RoboDK station: colorBars_ROR.rdk

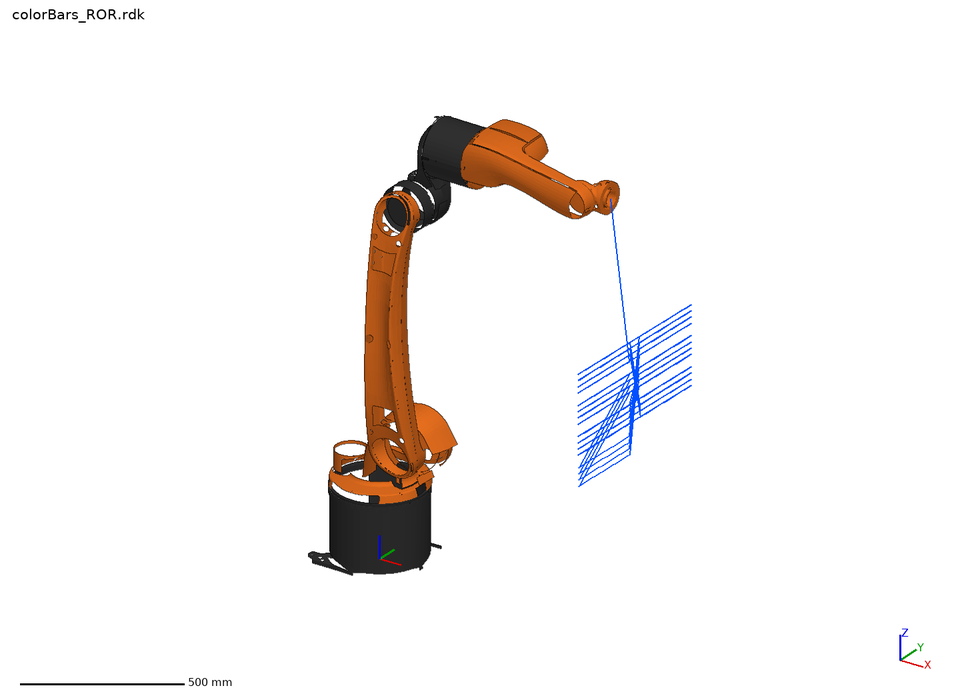
[picture v0: the station drawn from its stored meshes, robots at their saved joint values, targets as dots, program paths as lines]
Station pv_f053_run_on_robot (saved by RoboDK 5.4.1). Poses are relative to the parent item; angles as X-Y-Z fixed-axis rotations.
  - frame KR 8 1620 ARC HW Base at (0, 0, 0) mm
    - robot KR 8 1620 ARC HW: 6 axes
        modified DH rows (alpha deg, a mm, theta deg, d mm): 0, 0, 0, 450; -90, 150, 0, 0; 0, 810, -90, 0; -90, 200, 0, 630; 90, 0, 0, 0; -90, 0, 180, 80
        joint limits [-170, -185, -120, -165, -115, -350] to [170, 65, 180, 165, 140, 350]; home [0, -90, 90, 0, 0, 0]; saved at [0, -90, 90, 0, 0, 0]
      - tool fbx_0_slot_00_fo1_roundShape_outPaintBrush, TCP at (-4.14, -15.45, 32) mm
      - tool fbx_1_slot_01_fo2_roundShape_outPaintBrush, TCP at (-15.45, -4.14, 32) mm
      - tool fbx_2_slot_02_fo3_roundShape_outPaintBrush, TCP at (-11.31, 11.31, 32) mm
      - tool fbx_3_slot_03_fo4_roundShape_outPaintBrush, TCP at (4.14, 15.45, 32) mm
      - tool fbx_4_slot_04_fo5_roundShape_outPaintBrush, TCP at (15.45, 4.14, 32) mm
      - tool fbx_5_slot_05_fo6_roundShape_outPaintBrush, TCP at (11.31, -11.31, 32) mm
  - frame ax_frame at (0, 0, 0) mm
    - target home_approach (joint target) at (860, 0, 1460) mm, rotated rx 0 ry 90 rz 0 deg; joints [0, -89.818, 101.483, 0, -11.665, 0] of KR 8 1620 ARC HW
  - program pv_f053_00 (1123 instructions, listed below)
  - frame pv_f053_00_frame at (0, 0, 0) mm
    - target init_t0 (Cartesian target) at (979.8, -18.27, 823.95) mm, rotated rx 136.82 ry 86.87 rz 134.63 deg; joints [1.647, -75.367, 132.098, -0.612, -54.447, -1.81] of KR 8 1620 ARC HW
    - target stk_p0_s0_t0 (Cartesian target) at (979.8, -18.27, 823.95) mm, rotated rx 136.82 ry 86.87 rz 134.63 deg; joints [1.647, -75.367, 132.098, -0.612, -54.447, -1.81] of KR 8 1620 ARC HW
    - target stk_p0_s0_t0 (Cartesian target) at (979.8, -18.27, 823.95) mm, rotated rx 136.82 ry 86.87 rz 134.63 deg; joints [1.647, -75.367, 132.098, -0.612, -54.447, -1.81] of KR 8 1620 ARC HW
    - target stk_p0_s0_t1 (Cartesian target) at (980.02, -7.71, 824.07) mm, rotated rx 132.07 ry 86.58 rz 129.48 deg; joints [0.893, -75.374, 132.102, -2.02, -54.454, -1.429] of KR 8 1620 ARC HW
    - target stk_p0_s0_t2 (Cartesian target) at (980.24, 2.85, 824.19) mm, rotated rx 128.07 ry 86.28 rz 125.08 deg; joints [0.139, -75.372, 132.093, -3.428, -54.473, -1.049] of KR 8 1620 ARC HW
    - target stk_p0_s0_t3 (Cartesian target) at (980.46, 13.4, 824.32) mm, rotated rx 124.68 ry 85.96 rz 121.29 deg; joints [-0.614, -75.361, 132.07, -4.835, -54.503, -0.67] of KR 8 1620 ARC HW
    - target stk_p0_s0_t4 (Cartesian target) at (980.68, 23.96, 824.44) mm, rotated rx 121.8 ry 85.63 rz 118.01 deg; joints [-1.367, -75.34, 132.034, -6.239, -54.545, -0.292] of KR 8 1620 ARC HW
    - target stk_p0_s0_t5 (Cartesian target) at (980.89, 34.52, 824.56) mm, rotated rx 119.33 ry 85.29 rz 115.14 deg; joints [-2.12, -75.31, 131.985, -7.642, -54.598, 0.085] of KR 8 1620 ARC HW
    - target stk_p0_s0_t6 (Cartesian target) at (981.11, 45.08, 824.69) mm, rotated rx 117.2 ry 84.94 rz 112.61 deg; joints [-2.871, -75.27, 131.923, -9.04, -54.663, 0.46] of KR 8 1620 ARC HW
    - target stk_p0_s0_t7 (Cartesian target) at (981.33, 55.64, 824.81) mm, rotated rx 115.34 ry 84.59 rz 110.35 deg; joints [-3.621, -75.221, 131.848, -10.435, -54.74, 0.832] of KR 8 1620 ARC HW
    - target stk_p0_s0_t8 (Cartesian target) at (981.55, 66.2, 824.94) mm, rotated rx 113.72 ry 84.23 rz 108.33 deg; joints [-4.369, -75.163, 131.759, -11.825, -54.828, 1.201] of KR 8 1620 ARC HW
    - target stk_p0_s0_t9 (Cartesian target) at (981.77, 76.75, 825.06) mm, rotated rx 112.28 ry 83.87 rz 106.49 deg; joints [-5.115, -75.095, 131.658, -13.21, -54.927, 1.567] of KR 8 1620 ARC HW
    - target stk_p0_s0_t10 (Cartesian target) at (981.99, 87.31, 825.18) mm, rotated rx 111.01 ry 83.51 rz 104.82 deg; joints [-5.859, -75.019, 131.543, -14.588, -55.037, 1.929] of KR 8 1620 ARC HW
    - target stk_p0_s0_t11 (Cartesian target) at (982.21, 97.87, 825.31) mm, rotated rx 109.87 ry 83.14 rz 103.28 deg; joints [-6.601, -74.933, 131.415, -15.961, -55.158, 2.288] of KR 8 1620 ARC HW
    - target stk_p0_s0_t12 (Cartesian target) at (982.43, 108.43, 825.43) mm, rotated rx 108.85 ry 82.77 rz 101.87 deg; joints [-7.339, -74.838, 131.274, -17.325, -55.289, 2.642] of KR 8 1620 ARC HW
    - target stk_p0_s0_t13 (Cartesian target) at (982.65, 118.99, 825.55) mm, rotated rx 107.93 ry 82.4 rz 100.55 deg; joints [-8.075, -74.733, 131.12, -18.682, -55.431, 2.991] of KR 8 1620 ARC HW
    - target stk_p0_s0_t14 (Cartesian target) at (982.87, 129.55, 825.68) mm, rotated rx 107.09 ry 82.03 rz 99.32 deg; joints [-8.808, -74.62, 130.953, -20.031, -55.583, 3.336] of KR 8 1620 ARC HW
    - target stk_p0_s0_t15 (Cartesian target) at (983.09, 140.11, 825.8) mm, rotated rx 106.33 ry 81.66 rz 98.16 deg; joints [-9.537, -74.498, 130.773, -21.371, -55.745, 3.675] of KR 8 1620 ARC HW
    - target stk_p0_s0_t16 (Cartesian target) at (983.31, 150.66, 825.92) mm, rotated rx 105.64 ry 81.29 rz 97.07 deg; joints [-10.262, -74.367, 130.58, -22.701, -55.917, 4.009] of KR 8 1620 ARC HW
    - target stk_p0_s0_t17 (Cartesian target) at (983.53, 161.22, 826.05) mm, rotated rx 105 ry 80.91 rz 96.04 deg; joints [-10.984, -74.228, 130.374, -24.022, -56.098, 4.338] of KR 8 1620 ARC HW
    - target stk_p0_s0_t18 (Cartesian target) at (983.75, 171.78, 826.17) mm, rotated rx 104.42 ry 80.54 rz 95.06 deg; joints [-11.701, -74.08, 130.155, -25.332, -56.289, 4.66] of KR 8 1620 ARC HW
    - target stk_p0_s0_t19 (Cartesian target) at (983.96, 182.34, 826.29) mm, rotated rx 103.88 ry 80.17 rz 94.13 deg; joints [-12.414, -73.923, 129.923, -26.632, -56.488, 4.977] of KR 8 1620 ARC HW
    - target stk_p0_s0_t20 (Cartesian target) at (984.18, 192.9, 826.42) mm, rotated rx 103.38 ry 79.79 rz 93.24 deg; joints [-13.123, -73.758, 129.679, -27.92, -56.696, 5.288] of KR 8 1620 ARC HW
    - target stk_p0_s0_t21 (Cartesian target) at (984.4, 203.46, 826.54) mm, rotated rx 102.91 ry 79.42 rz 92.38 deg; joints [-13.826, -73.584, 129.422, -29.198, -56.912, 5.593] of KR 8 1620 ARC HW
    - target stk_p0_s0_t22 (Cartesian target) at (984.62, 214.01, 826.67) mm, rotated rx 102.48 ry 79.05 rz 91.56 deg; joints [-14.525, -73.402, 129.152, -30.463, -57.136, 5.891] of KR 8 1620 ARC HW
    - target stk_p0_s0_t23 (Cartesian target) at (984.84, 224.57, 826.79) mm, rotated rx 102.08 ry 78.67 rz 90.76 deg; joints [-15.219, -73.212, 128.87, -31.717, -57.368, 6.183] of KR 8 1620 ARC HW
    - target stk_p0_s0_t24 (Cartesian target) at (985.06, 235.13, 826.91) mm, rotated rx 101.7 ry 78.3 rz 90 deg; joints [-15.907, -73.014, 128.575, -32.958, -57.608, 6.469] of KR 8 1620 ARC HW
    - target stk_p0_s0_t25 (Cartesian target) at (985.28, 245.69, 827.04) mm, rotated rx 101.35 ry 77.93 rz 89.26 deg; joints [-16.59, -72.808, 128.268, -34.186, -57.855, 6.749] of KR 8 1620 ARC HW
    - target stk_p0_s1_t0 (Cartesian target) at (973.22, -335.02, 820.24) mm, rotated rx -102.56 ry 80.25 rz -92.87 deg; joints [22.967, -71.014, 125.959, 38.741, -59.048, -11.564] of KR 8 1620 ARC HW
    - target stk_p0_s1_t0 (Cartesian target) at (973.22, -335.02, 820.24) mm, rotated rx -102.56 ry 80.25 rz -92.87 deg; joints [22.967, -71.014, 125.959, 38.741, -59.048, -11.564] of KR 8 1620 ARC HW
    - target stk_p0_s1_t1 (Cartesian target) at (973.44, -324.47, 820.36) mm, rotated rx -103.11 ry 80.62 rz -93.8 deg; joints [22.327, -71.275, 126.345, 37.585, -58.778, -11.319] of KR 8 1620 ARC HW
    - target stk_p0_s1_t2 (Cartesian target) at (973.66, -313.91, 820.49) mm, rotated rx -103.7 ry 80.99 rz -94.78 deg; joints [21.681, -71.529, 126.719, 36.415, -58.514, -11.068] of KR 8 1620 ARC HW
    - target stk_p0_s1_t3 (Cartesian target) at (973.88, -303.35, 820.61) mm, rotated rx -104.33 ry 81.36 rz -95.8 deg; joints [21.028, -71.776, 127.08, 35.233, -58.255, -10.811] of KR 8 1620 ARC HW
    - target stk_p0_s1_t4 (Cartesian target) at (974.1, -292.79, 820.73) mm, rotated rx -105.03 ry 81.73 rz -96.89 deg; joints [20.37, -72.016, 127.43, 34.037, -58.003, -10.548] of KR 8 1620 ARC HW
    - target stk_p0_s1_t5 (Cartesian target) at (974.32, -282.23, 820.86) mm, rotated rx -105.8 ry 82.1 rz -98.05 deg; joints [19.705, -72.248, 127.767, 32.829, -57.757, -10.279] of KR 8 1620 ARC HW
    - target stk_p0_s1_t6 (Cartesian target) at (974.53, -271.67, 820.98) mm, rotated rx -106.64 ry 82.46 rz -99.28 deg; joints [19.035, -72.474, 128.093, 31.608, -57.517, -10.004] of KR 8 1620 ARC HW
    - target stk_p0_s1_t7 (Cartesian target) at (974.75, -261.11, 821.11) mm, rotated rx -107.56 ry 82.83 rz -100.59 deg; joints [18.359, -72.691, 128.406, 30.375, -57.285, -9.722] of KR 8 1620 ARC HW
    - target stk_p0_s1_t8 (Cartesian target) at (974.97, -250.56, 821.23) mm, rotated rx -108.59 ry 83.19 rz -102.01 deg; joints [17.677, -72.901, 128.706, 29.129, -57.059, -9.435] of KR 8 1620 ARC HW
    - target stk_p0_s1_t9 (Cartesian target) at (975.19, -240, 821.35) mm, rotated rx -109.73 ry 83.56 rz -103.55 deg; joints [16.99, -73.103, 128.995, 27.872, -56.841, -9.142] of KR 8 1620 ARC HW
    - target stk_p0_s1_t10 (Cartesian target) at (975.41, -229.44, 821.48) mm, rotated rx -111.02 ry 83.92 rz -105.23 deg; joints [16.297, -73.297, 129.271, 26.602, -56.631, -8.842] of KR 8 1620 ARC HW
    - target stk_p0_s1_t11 (Cartesian target) at (975.63, -218.88, 821.6) mm, rotated rx -112.46 ry 84.28 rz -107.07 deg; joints [15.6, -73.483, 129.534, 25.321, -56.429, -8.536] of KR 8 1620 ARC HW
    - target stk_p0_s1_t12 (Cartesian target) at (975.85, -208.32, 821.72) mm, rotated rx -114.1 ry 84.63 rz -109.1 deg; joints [14.897, -73.661, 129.785, 24.029, -56.235, -8.224] of KR 8 1620 ARC HW
    - target stk_p0_s1_t13 (Cartesian target) at (976.07, -197.76, 821.85) mm, rotated rx -115.97 ry 84.98 rz -111.37 deg; joints [14.19, -73.83, 130.023, 22.726, -56.05, -7.907] of KR 8 1620 ARC HW
    - target stk_p0_s1_t14 (Cartesian target) at (976.29, -187.21, 821.97) mm, rotated rx -118.12 ry 85.32 rz -113.92 deg; joints [13.478, -73.992, 130.249, 21.413, -55.874, -7.583] of KR 8 1620 ARC HW
    - target stk_p0_s1_t15 (Cartesian target) at (976.51, -176.65, 822.09) mm, rotated rx -120.61 ry 85.66 rz -116.81 deg; joints [12.762, -74.144, 130.461, 20.089, -55.707, -7.254] of KR 8 1620 ARC HW
    - target stk_p0_s1_t16 (Cartesian target) at (976.73, -166.09, 822.22) mm, rotated rx -123.52 ry 85.99 rz -120.11 deg; joints [12.041, -74.289, 130.662, 18.756, -55.549, -6.919] of KR 8 1620 ARC HW
    - target stk_p0_s1_t17 (Cartesian target) at (976.95, -155.53, 822.34) mm, rotated rx -126.94 ry 86.3 rz -123.92 deg; joints [11.317, -74.424, 130.849, 17.414, -55.4, -6.579] of KR 8 1620 ARC HW
    - target stk_p0_s1_t18 (Cartesian target) at (977.17, -144.97, 822.46) mm, rotated rx -130.98 ry 86.61 rz -128.36 deg; joints [10.589, -74.551, 131.023, 16.063, -55.262, -6.234] of KR 8 1620 ARC HW
    - target stk_p0_s1_t19 (Cartesian target) at (977.39, -134.41, 822.59) mm, rotated rx -135.78 ry 86.89 rz -133.56 deg; joints [9.857, -74.67, 131.185, 14.704, -55.134, -5.883] of KR 8 1620 ARC HW
    - target stk_p0_s1_t20 (Cartesian target) at (977.6, -123.86, 822.71) mm, rotated rx -141.48 ry 87.14 rz -139.67 deg; joints [9.122, -74.779, 131.333, 13.337, -55.016, -5.529] of KR 8 1620 ARC HW
    - target stk_p0_s1_t21 (Cartesian target) at (977.82, -113.3, 822.84) mm, rotated rx -148.23 ry 87.36 rz -146.81 deg; joints [8.384, -74.879, 131.469, 11.964, -54.909, -5.17] of KR 8 1620 ARC HW
    - target stk_p0_s1_t22 (Cartesian target) at (978.04, -102.74, 822.96) mm, rotated rx -156.09 ry 87.54 rz -155.07 deg; joints [7.643, -74.97, 131.591, 10.583, -54.812, -4.807] of KR 8 1620 ARC HW
    - target stk_p0_s1_t23 (Cartesian target) at (978.26, -92.18, 823.08) mm, rotated rx -164.99 ry 87.67 rz -164.37 deg; joints [6.899, -75.052, 131.7, 9.197, -54.727, -4.441] of KR 8 1620 ARC HW
    - target stk_p0_s1_t24 (Cartesian target) at (978.48, -81.62, 823.21) mm, rotated rx -174.64 ry 87.73 rz -174.43 deg; joints [6.154, -75.125, 131.797, 7.806, -54.653, -4.071] of KR 8 1620 ARC HW
    - target stk_p0_s1_t25 (Cartesian target) at (978.7, -71.06, 823.33) mm, rotated rx 175.43 ry 87.73 rz 175.24 deg; joints [5.406, -75.189, 131.88, 6.41, -54.59, -3.699] of KR 8 1620 ARC HW
    - target stk_p0_s2_t0 (Cartesian target) at (979.98, -19.51, 929.55) mm, rotated rx 161.34 ry 83.46 rz 159.13 deg; joints [1.735, -80.185, 126.571, -0.562, -40.195, -1.71] of KR 8 1620 ARC HW
    - target stk_p0_s2_t0 (Cartesian target) at (979.98, -19.51, 929.55) mm, rotated rx 161.34 ry 83.46 rz 159.13 deg; joints [1.735, -80.185, 126.571, -0.562, -40.195, -1.71] of KR 8 1620 ARC HW
    - target stk_p0_s2_t1 (Cartesian target) at (980.2, -8.95, 929.68) mm, rotated rx 158.17 ry 83.32 rz 155.54 deg; joints [0.981, -80.194, 126.576, -2.328, -40.208, -0.877] of KR 8 1620 ARC HW
    - target stk_p0_s2_t2 (Cartesian target) at (980.42, 1.61, 929.8) mm, rotated rx 155.13 ry 83.16 rz 152.09 deg; joints [0.227, -80.192, 126.568, -4.093, -40.243, -0.046] of KR 8 1620 ARC HW
    - target stk_p0_s2_t3 (Cartesian target) at (980.64, 12.16, 929.92) mm, rotated rx 152.25 ry 82.99 rz 148.79 deg; joints [-0.527, -80.18, 126.548, -5.854, -40.3, 0.782] of KR 8 1620 ARC HW
    - target stk_p0_s2_t4 (Cartesian target) at (980.86, 22.72, 930.05) mm, rotated rx 149.51 ry 82.79 rz 145.64 deg; joints [-1.28, -80.158, 126.515, -7.61, -40.379, 1.605] of KR 8 1620 ARC HW
    - target stk_p0_s2_t5 (Cartesian target) at (981.08, 33.28, 930.17) mm, rotated rx 146.92 ry 82.59 rz 142.64 deg; joints [-2.033, -80.126, 126.469, -9.358, -40.48, 2.421] of KR 8 1620 ARC HW
    - target stk_p0_s2_t6 (Cartesian target) at (981.3, 43.84, 930.3) mm, rotated rx 144.48 ry 82.36 rz 139.79 deg; joints [-2.784, -80.083, 126.41, -11.097, -40.602, 3.229] of KR 8 1620 ARC HW
    - target stk_p0_s2_t7 (Cartesian target) at (981.52, 54.4, 930.42) mm, rotated rx 142.18 ry 82.13 rz 137.08 deg; joints [-3.535, -80.03, 126.339, -12.826, -40.745, 4.027] of KR 8 1620 ARC HW
    - target stk_p0_s2_t8 (Cartesian target) at (981.74, 64.96, 930.54) mm, rotated rx 140.02 ry 81.88 rz 134.5 deg; joints [-4.283, -79.967, 126.255, -14.541, -40.909, 4.814] of KR 8 1620 ARC HW
    - target stk_p0_s2_t9 (Cartesian target) at (981.96, 75.52, 930.67) mm, rotated rx 138 ry 81.62 rz 132.06 deg; joints [-5.03, -79.894, 126.158, -16.243, -41.094, 5.589] of KR 8 1620 ARC HW
    - target stk_p0_s2_t10 (Cartesian target) at (982.18, 86.07, 930.79) mm, rotated rx 136.09 ry 81.36 rz 129.75 deg; joints [-5.774, -79.81, 126.049, -17.929, -41.299, 6.349] of KR 8 1620 ARC HW
    - target stk_p0_s2_t11 (Cartesian target) at (982.39, 96.63, 930.91) mm, rotated rx 134.3 ry 81.08 rz 127.55 deg; joints [-6.516, -79.717, 125.927, -19.598, -41.522, 7.094] of KR 8 1620 ARC HW
    - target stk_p0_s2_t12 (Cartesian target) at (982.61, 107.19, 931.04) mm, rotated rx 132.63 ry 80.8 rz 125.46 deg; joints [-7.256, -79.614, 125.792, -21.249, -41.765, 7.824] of KR 8 1620 ARC HW
    - target stk_p0_s2_t13 (Cartesian target) at (982.83, 117.75, 931.16) mm, rotated rx 131.05 ry 80.51 rz 123.47 deg; joints [-7.992, -79.501, 125.645, -22.88, -42.026, 8.536] of KR 8 1620 ARC HW
    - target stk_p0_s2_t14 (Cartesian target) at (983.05, 128.31, 931.28) mm, rotated rx 129.57 ry 80.21 rz 121.58 deg; joints [-8.725, -79.378, 125.485, -24.492, -42.304, 9.23] of KR 8 1620 ARC HW
    - target stk_p0_s2_t15 (Cartesian target) at (983.27, 138.87, 931.41) mm, rotated rx 128.18 ry 79.91 rz 119.78 deg; joints [-9.455, -79.245, 125.312, -26.082, -42.6, 9.906] of KR 8 1620 ARC HW
    - target stk_p0_s2_t16 (Cartesian target) at (983.49, 149.42, 931.53) mm, rotated rx 126.87 ry 79.6 rz 118.07 deg; joints [-10.181, -79.103, 125.127, -27.649, -42.911, 10.563] of KR 8 1620 ARC HW
    - target stk_p0_s2_t17 (Cartesian target) at (983.71, 159.98, 931.65) mm, rotated rx 125.64 ry 79.29 rz 116.43 deg; joints [-10.904, -78.951, 124.929, -29.194, -43.238, 11.2] of KR 8 1620 ARC HW
    - target stk_p0_s2_t18 (Cartesian target) at (983.93, 170.54, 931.78) mm, rotated rx 124.48 ry 78.98 rz 114.86 deg; joints [-11.622, -78.79, 124.719, -30.716, -43.58, 11.817] of KR 8 1620 ARC HW
    - target stk_p0_s2_t19 (Cartesian target) at (984.15, 181.1, 931.9) mm, rotated rx 123.39 ry 78.66 rz 113.36 deg; joints [-12.336, -78.62, 124.496, -32.214, -43.936, 12.413] of KR 8 1620 ARC HW
    - target stk_p0_s2_t20 (Cartesian target) at (984.37, 191.66, 932.02) mm, rotated rx 122.36 ry 78.34 rz 111.93 deg; joints [-13.045, -78.44, 124.261, -33.688, -44.305, 12.99] of KR 8 1620 ARC HW
    - target stk_p0_s2_t21 (Cartesian target) at (984.59, 202.22, 932.15) mm, rotated rx 121.38 ry 78.01 rz 110.55 deg; joints [-13.749, -78.251, 124.014, -35.138, -44.687, 13.546] of KR 8 1620 ARC HW
    - target stk_p0_s2_t22 (Cartesian target) at (984.81, 212.77, 932.27) mm, rotated rx 120.46 ry 77.68 rz 109.22 deg; joints [-14.449, -78.054, 123.754, -36.563, -45.081, 14.082] of KR 8 1620 ARC HW
    - target stk_p0_s2_t23 (Cartesian target) at (985.03, 223.33, 932.4) mm, rotated rx 119.58 ry 77.35 rz 107.94 deg; joints [-15.143, -77.847, 123.482, -37.964, -45.487, 14.597] of KR 8 1620 ARC HW
    - target stk_p0_s2_t24 (Cartesian target) at (985.25, 233.89, 932.52) mm, rotated rx 118.76 ry 77.02 rz 106.71 deg; joints [-15.833, -77.632, 123.197, -39.34, -45.903, 15.093] of KR 8 1620 ARC HW
    - target stk_p0_s2_t25 (Cartesian target) at (985.46, 244.45, 932.64) mm, rotated rx 117.97 ry 76.69 rz 105.53 deg; joints [-16.516, -77.408, 122.9, -40.691, -46.329, 15.568] of KR 8 1620 ARC HW
    - target stk_p0_s3_t0 (Cartesian target) at (973.4, -336.26, 925.85) mm, rotated rx -122.11 ry 78.75 rz -112.05 deg; joints [23.04, -75.435, 120.599, 45.803, -48.371, -20.985] of KR 8 1620 ARC HW
    - target stk_p0_s3_t0 (Cartesian target) at (973.4, -336.26, 925.85) mm, rotated rx -122.11 ry 78.75 rz -112.05 deg; joints [23.04, -75.435, 120.599, 45.803, -48.371, -20.985] of KR 8 1620 ARC HW
    - target stk_p0_s3_t1 (Cartesian target) at (973.62, -325.7, 925.97) mm, rotated rx -123.2 ry 79.07 rz -113.54 deg; joints [22.401, -75.719, 120.975, 44.576, -47.917, -20.603] of KR 8 1620 ARC HW
    - target stk_p0_s3_t2 (Cartesian target) at (973.84, -315.15, 926.09) mm, rotated rx -124.37 ry 79.38 rz -115.11 deg; joints [21.755, -75.996, 121.339, 43.326, -47.469, -20.204] of KR 8 1620 ARC HW
    - target stk_p0_s3_t3 (Cartesian target) at (974.06, -304.59, 926.22) mm, rotated rx -125.6 ry 79.68 rz -116.74 deg; joints [21.104, -76.265, 121.692, 42.053, -47.028, -19.787] of KR 8 1620 ARC HW
    - target stk_p0_s3_t4 (Cartesian target) at (974.28, -294.03, 926.34) mm, rotated rx -126.92 ry 79.98 rz -118.46 deg; joints [20.446, -76.526, 122.032, 40.756, -46.595, -19.352] of KR 8 1620 ARC HW
    - target stk_p0_s3_t5 (Cartesian target) at (974.5, -283.47, 926.47) mm, rotated rx -128.31 ry 80.28 rz -120.25 deg; joints [19.782, -76.779, 122.361, 39.434, -46.171, -18.899] of KR 8 1620 ARC HW
    - target stk_p0_s3_t6 (Cartesian target) at (974.72, -272.91, 926.59) mm, rotated rx -129.8 ry 80.57 rz -122.14 deg; joints [19.113, -77.025, 122.677, 38.089, -45.756, -18.426] of KR 8 1620 ARC HW
    - target stk_p0_s3_t7 (Cartesian target) at (974.94, -262.35, 926.71) mm, rotated rx -131.38 ry 80.86 rz -124.13 deg; joints [18.438, -77.262, 122.982, 36.72, -45.35, -17.934] of KR 8 1620 ARC HW
    - target stk_p0_s3_t8 (Cartesian target) at (975.16, -251.8, 926.84) mm, rotated rx -133.06 ry 81.14 rz -126.22 deg; joints [17.757, -77.49, 123.274, 35.326, -44.955, -17.422] of KR 8 1620 ARC HW
    - target stk_p0_s3_t9 (Cartesian target) at (975.38, -241.24, 926.96) mm, rotated rx -134.85 ry 81.41 rz -128.42 deg; joints [17.07, -77.711, 123.554, 33.907, -44.57, -16.89] of KR 8 1620 ARC HW
    - target stk_p0_s3_t10 (Cartesian target) at (975.6, -230.68, 927.08) mm, rotated rx -136.76 ry 81.67 rz -130.74 deg; joints [16.379, -77.922, 123.822, 32.464, -44.197, -16.338] of KR 8 1620 ARC HW
    - target stk_p0_s3_t11 (Cartesian target) at (975.82, -220.12, 927.21) mm, rotated rx -138.8 ry 81.93 rz -133.18 deg; joints [15.682, -78.125, 124.078, 30.997, -43.837, -15.766] of KR 8 1620 ARC HW
    - target stk_p0_s3_t12 (Cartesian target) at (976.03, -209.56, 927.33) mm, rotated rx -140.97 ry 82.17 rz -135.75 deg; joints [14.98, -78.319, 124.321, 29.507, -43.49, -15.174] of KR 8 1620 ARC HW
    - target stk_p0_s3_t13 (Cartesian target) at (976.25, -199, 927.45) mm, rotated rx -143.27 ry 82.4 rz -138.47 deg; joints [14.273, -78.504, 124.553, 27.992, -43.156, -14.561] of KR 8 1620 ARC HW
    - target stk_p0_s3_t14 (Cartesian target) at (976.47, -188.45, 927.58) mm, rotated rx -145.72 ry 82.62 rz -141.33 deg; joints [13.562, -78.68, 124.772, 26.454, -42.836, -13.929] of KR 8 1620 ARC HW
    - target stk_p0_s3_t15 (Cartesian target) at (976.69, -177.89, 927.7) mm, rotated rx -148.32 ry 82.82 rz -144.33 deg; joints [12.846, -78.847, 124.978, 24.893, -42.532, -13.277] of KR 8 1620 ARC HW
    - target stk_p0_s3_t16 (Cartesian target) at (976.91, -167.33, 927.82) mm, rotated rx -151.06 ry 83.02 rz -147.49 deg; joints [12.126, -79.005, 125.172, 23.31, -42.244, -12.607] of KR 8 1620 ARC HW
    - target stk_p0_s3_t17 (Cartesian target) at (977.13, -156.77, 927.95) mm, rotated rx -153.96 ry 83.19 rz -150.8 deg; joints [11.402, -79.153, 125.354, 21.706, -41.972, -11.917] of KR 8 1620 ARC HW
    - target stk_p0_s3_t18 (Cartesian target) at (977.35, -146.21, 928.07) mm, rotated rx -157 ry 83.34 rz -154.25 deg; joints [10.675, -79.292, 125.523, 20.081, -41.717, -11.21] of KR 8 1620 ARC HW
    - target stk_p0_s3_t19 (Cartesian target) at (977.57, -135.65, 928.19) mm, rotated rx -160.18 ry 83.48 rz -157.84 deg; joints [9.943, -79.421, 125.68, 18.437, -41.48, -10.485] of KR 8 1620 ARC HW
    - target stk_p0_s3_t20 (Cartesian target) at (977.79, -125.09, 928.32) mm, rotated rx -163.49 ry 83.6 rz -161.56 deg; joints [9.208, -79.54, 125.824, 16.774, -41.261, -9.744] of KR 8 1620 ARC HW
    - target stk_p0_s3_t21 (Cartesian target) at (978.01, -114.54, 928.44) mm, rotated rx -166.9 ry 83.69 rz -165.39 deg; joints [8.471, -79.65, 125.955, 15.093, -41.062, -8.988] of KR 8 1620 ARC HW
    - target stk_p0_s3_t22 (Cartesian target) at (978.23, -103.98, 928.57) mm, rotated rx -170.41 ry 83.76 rz -169.31 deg; joints [7.73, -79.75, 126.074, 13.397, -40.882, -8.218] of KR 8 1620 ARC HW
    - target stk_p0_s3_t23 (Cartesian target) at (978.45, -93.42, 928.69) mm, rotated rx -173.99 ry 83.81 rz -173.31 deg; joints [6.987, -79.839, 126.181, 11.686, -40.722, -7.434] of KR 8 1620 ARC HW
    - target stk_p0_s3_t24 (Cartesian target) at (978.67, -82.86, 928.81) mm, rotated rx -177.61 ry 83.83 rz -177.34 deg; joints [6.241, -79.919, 126.275, 9.962, -40.582, -6.639] of KR 8 1620 ARC HW
    - target stk_p0_s3_t25 (Cartesian target) at (978.89, -72.3, 928.94) mm, rotated rx 178.75 ry 83.83 rz 178.61 deg; joints [5.494, -79.989, 126.356, 8.226, -40.463, -5.834] of KR 8 1620 ARC HW
    - target stk_p0_s4_t0 (Cartesian target) at (973.03, -333.78, 714.63) mm, rotated rx -79.48 ry 80.37 rz -70.16 deg; joints [22.877, -65.289, 129.963, 34.563, -70.512, -4.58] of KR 8 1620 ARC HW
    - target stk_p0_s4_t0 (Cartesian target) at (973.03, -333.78, 714.63) mm, rotated rx -79.48 ry 80.37 rz -70.16 deg; joints [22.877, -65.289, 129.963, 34.563, -70.512, -4.58] of KR 8 1620 ARC HW
    - target stk_p0_s4_t1 (Cartesian target) at (973.25, -323.23, 714.76) mm, rotated rx -79.07 ry 80.74 rz -70.12 deg; joints [22.237, -65.517, 130.358, 33.479, -70.403, -4.479] of KR 8 1620 ARC HW
    - target stk_p0_s4_t2 (Cartesian target) at (973.47, -312.67, 714.88) mm, rotated rx -78.63 ry 81.12 rz -70.05 deg; joints [21.59, -65.739, 130.74, 32.387, -70.299, -4.38] of KR 8 1620 ARC HW
    - target stk_p0_s4_t3 (Cartesian target) at (973.69, -302.11, 715) mm, rotated rx -78.14 ry 81.49 rz -69.94 deg; joints [20.937, -65.955, 131.111, 31.287, -70.198, -4.281] of KR 8 1620 ARC HW
    - target stk_p0_s4_t4 (Cartesian target) at (973.91, -291.55, 715.13) mm, rotated rx -77.61 ry 81.87 rz -69.79 deg; joints [20.278, -66.165, 131.469, 30.179, -70.1, -4.184] of KR 8 1620 ARC HW
    - target stk_p0_s4_t5 (Cartesian target) at (974.13, -280.99, 715.25) mm, rotated rx -77.03 ry 82.24 rz -69.58 deg; joints [19.613, -66.367, 131.815, 29.064, -70.006, -4.089] of KR 8 1620 ARC HW
    - target stk_p0_s4_t6 (Cartesian target) at (974.35, -270.43, 715.38) mm, rotated rx -76.38 ry 82.62 rz -69.31 deg; joints [18.942, -66.563, 132.148, 27.94, -69.915, -3.994] of KR 8 1620 ARC HW
    - target stk_p0_s4_t7 (Cartesian target) at (974.57, -259.88, 715.5) mm, rotated rx -75.67 ry 82.99 rz -68.98 deg; joints [18.266, -66.753, 132.469, 26.809, -69.828, -3.901] of KR 8 1620 ARC HW
    - target stk_p0_s4_t8 (Cartesian target) at (974.79, -249.32, 715.62) mm, rotated rx -74.87 ry 83.36 rz -68.56 deg; joints [17.584, -66.935, 132.778, 25.671, -69.745, -3.809] of KR 8 1620 ARC HW
    - target stk_p0_s4_t9 (Cartesian target) at (975.01, -238.76, 715.75) mm, rotated rx -73.98 ry 83.74 rz -68.05 deg; joints [16.897, -67.111, 133.074, 24.525, -69.665, -3.718] of KR 8 1620 ARC HW
    - target stk_p0_s4_t10 (Cartesian target) at (975.23, -228.2, 715.87) mm, rotated rx -72.97 ry 84.11 rz -67.43 deg; joints [16.204, -67.279, 133.357, 23.373, -69.588, -3.628] of KR 8 1620 ARC HW
    - target stk_p0_s4_t11 (Cartesian target) at (975.45, -217.64, 715.99) mm, rotated rx -71.83 ry 84.48 rz -66.67 deg; joints [15.506, -67.441, 133.628, 22.215, -69.515, -3.538] of KR 8 1620 ARC HW
    - target stk_p0_s4_t12 (Cartesian target) at (975.67, -207.08, 716.12) mm, rotated rx -70.52 ry 84.85 rz -65.74 deg; joints [14.804, -67.595, 133.885, 21.05, -69.446, -3.45] of KR 8 1620 ARC HW
    - target stk_p0_s4_t13 (Cartesian target) at (975.89, -196.52, 716.24) mm, rotated rx -69.01 ry 85.21 rz -64.61 deg; joints [14.096, -67.742, 134.13, 19.878, -69.38, -3.362] of KR 8 1620 ARC HW
    - target stk_p0_s4_t14 (Cartesian target) at (976.1, -185.97, 716.36) mm, rotated rx -67.25 ry 85.58 rz -63.24 deg; joints [13.384, -67.882, 134.362, 18.701, -69.318, -3.275] of KR 8 1620 ARC HW
    - target stk_p0_s4_t15 (Cartesian target) at (976.32, -175.41, 716.49) mm, rotated rx -65.18 ry 85.94 rz -61.54 deg; joints [12.668, -68.015, 134.58, 17.519, -69.26, -3.189] of KR 8 1620 ARC HW
    - target stk_p0_s4_t16 (Cartesian target) at (976.54, -164.85, 716.61) mm, rotated rx -62.7 ry 86.29 rz -59.45 deg; joints [11.947, -68.14, 134.786, 16.331, -69.205, -3.103] of KR 8 1620 ARC HW
    - target stk_p0_s4_t17 (Cartesian target) at (976.76, -154.29, 716.73) mm, rotated rx -59.72 ry 86.63 rz -56.85 deg; joints [11.223, -68.257, 134.978, 15.138, -69.154, -3.017] of KR 8 1620 ARC HW
    - target stk_p0_s4_t18 (Cartesian target) at (976.98, -143.73, 716.86) mm, rotated rx -56.06 ry 86.97 rz -53.57 deg; joints [10.495, -68.367, 135.157, 13.941, -69.106, -2.932] of KR 8 1620 ARC HW
    - target stk_p0_s4_t19 (Cartesian target) at (977.2, -133.17, 716.98) mm, rotated rx -51.51 ry 87.28 rz -49.42 deg; joints [9.764, -68.469, 135.323, 12.739, -69.062, -2.848] of KR 8 1620 ARC HW
    - target stk_p0_s4_t20 (Cartesian target) at (977.42, -122.62, 717.1) mm, rotated rx -45.81 ry 87.58 rz -44.1 deg; joints [9.029, -68.563, 135.476, 11.533, -69.022, -2.764] of KR 8 1620 ARC HW
    - target stk_p0_s4_t21 (Cartesian target) at (977.64, -112.06, 717.23) mm, rotated rx -38.59 ry 87.85 rz -37.27 deg; joints [8.291, -68.65, 135.615, 10.323, -68.986, -2.68] of KR 8 1620 ARC HW
    - target stk_p0_s4_t22 (Cartesian target) at (977.86, -101.5, 717.35) mm, rotated rx -29.53 ry 88.07 rz -28.59 deg; joints [7.551, -68.728, 135.74, 9.11, -68.953, -2.596] of KR 8 1620 ARC HW
    - target stk_p0_s4_t23 (Cartesian target) at (978.08, -90.94, 717.48) mm, rotated rx -18.44 ry 88.24 rz -17.89 deg; joints [6.808, -68.799, 135.852, 7.894, -68.924, -2.512] of KR 8 1620 ARC HW
    - target stk_p0_s4_t24 (Cartesian target) at (978.3, -80.38, 717.6) mm, rotated rx -5.66 ry 88.32 rz -5.5 deg; joints [6.062, -68.862, 135.951, 6.675, -68.899, -2.429] of KR 8 1620 ARC HW
    - target stk_p0_s4_t25 (Cartesian target) at (978.52, -69.82, 717.72) mm, rotated rx 7.77 ry 88.32 rz 7.54 deg; joints [5.315, -68.917, 136.036, 5.453, -68.878, -2.346] of KR 8 1620 ARC HW
    - target stk_p0_s5_t0 (Cartesian target) at (980.17, -20.75, 1035.16) mm, rotated rx 168.56 ry 79.75 rz 166.32 deg; joints [1.823, -83.495, 119.78, -0.514, -26.243, -1.633] of KR 8 1620 ARC HW
    - target stk_p0_s5_t0 (Cartesian target) at (980.17, -20.75, 1035.16) mm, rotated rx 168.56 ry 79.75 rz 166.32 deg; joints [1.823, -83.495, 119.78, -0.514, -26.243, -1.633] of KR 8 1620 ARC HW
    - target stk_p0_s5_t1 (Cartesian target) at (980.39, -10.19, 1035.28) mm, rotated rx 166.45 ry 79.66 rz 163.79 deg; joints [1.07, -83.504, 119.786, -3.065, -26.265, 0.062] of KR 8 1620 ARC HW
    - target stk_p0_s5_t2 (Cartesian target) at (980.6, 0.37, 1035.41) mm, rotated rx 164.38 ry 79.56 rz 161.29 deg; joints [0.316, -83.503, 119.78, -5.61, -26.327, 1.751] of KR 8 1620 ARC HW
    - target stk_p0_s5_t3 (Cartesian target) at (980.82, 10.93, 1035.53) mm, rotated rx 162.35 ry 79.45 rz 158.84 deg; joints [-0.437, -83.492, 119.761, -8.139, -26.429, 3.425] of KR 8 1620 ARC HW
    - target stk_p0_s5_t4 (Cartesian target) at (981.04, 21.48, 1035.65) mm, rotated rx 160.37 ry 79.32 rz 156.43 deg; joints [-1.19, -83.469, 119.73, -10.648, -26.569, 5.078] of KR 8 1620 ARC HW
    - target stk_p0_s5_t5 (Cartesian target) at (981.26, 32.04, 1035.78) mm, rotated rx 158.44 ry 79.18 rz 154.07 deg; joints [-1.942, -83.436, 119.687, -13.128, -26.748, 6.704] of KR 8 1620 ARC HW
    - target stk_p0_s5_t6 (Cartesian target) at (981.48, 42.6, 1035.9) mm, rotated rx 156.56 ry 79.03 rz 151.76 deg; joints [-2.694, -83.392, 119.631, -15.574, -26.965, 8.296] of KR 8 1620 ARC HW
    - target stk_p0_s5_t7 (Cartesian target) at (981.7, 53.16, 1036.03) mm, rotated rx 154.74 ry 78.87 rz 149.51 deg; joints [-3.443, -83.337, 119.564, -17.98, -27.218, 9.849] of KR 8 1620 ARC HW
    - target stk_p0_s5_t8 (Cartesian target) at (981.92, 63.72, 1036.15) mm, rotated rx 152.96 ry 78.7 rz 147.32 deg; joints [-4.192, -83.272, 119.484, -20.341, -27.506, 11.358] of KR 8 1620 ARC HW
    - target stk_p0_s5_t9 (Cartesian target) at (982.14, 74.28, 1036.27) mm, rotated rx 151.25 ry 78.51 rz 145.17 deg; joints [-4.938, -83.196, 119.391, -22.653, -27.827, 12.819] of KR 8 1620 ARC HW
    - target stk_p0_s5_t10 (Cartesian target) at (982.36, 84.83, 1036.4) mm, rotated rx 149.59 ry 78.32 rz 143.09 deg; joints [-5.683, -83.11, 119.287, -24.913, -28.181, 14.228] of KR 8 1620 ARC HW
    - target stk_p0_s5_t11 (Cartesian target) at (982.58, 95.39, 1036.52) mm, rotated rx 147.99 ry 78.12 rz 141.06 deg; joints [-6.425, -83.013, 119.17, -27.117, -28.565, 15.584] of KR 8 1620 ARC HW
    - target stk_p0_s5_t12 (Cartesian target) at (982.8, 105.95, 1036.64) mm, rotated rx 146.44 ry 77.91 rz 139.09 deg; joints [-7.164, -82.905, 119.04, -29.264, -28.978, 16.884] of KR 8 1620 ARC HW
    - target stk_p0_s5_t13 (Cartesian target) at (983.02, 116.51, 1036.77) mm, rotated rx 144.94 ry 77.69 rz 137.17 deg; joints [-7.9, -82.788, 118.899, -31.351, -29.418, 18.127] of KR 8 1620 ARC HW
    - target stk_p0_s5_t14 (Cartesian target) at (983.24, 127.07, 1036.89) mm, rotated rx 143.51 ry 77.47 rz 135.31 deg; joints [-8.634, -82.66, 118.745, -33.379, -29.884, 19.312] of KR 8 1620 ARC HW
    - target stk_p0_s5_t15 (Cartesian target) at (983.46, 137.63, 1037.01) mm, rotated rx 142.12 ry 77.24 rz 133.5 deg; joints [-9.364, -82.522, 118.579, -35.346, -30.374, 20.439] of KR 8 1620 ARC HW
    - target stk_p0_s5_t16 (Cartesian target) at (983.68, 148.18, 1037.14) mm, rotated rx 140.78 ry 77 rz 131.75 deg; joints [-10.09, -82.374, 118.401, -37.254, -30.887, 21.507] of KR 8 1620 ARC HW
    - target stk_p0_s5_t17 (Cartesian target) at (983.89, 158.74, 1037.26) mm, rotated rx 139.5 ry 76.75 rz 130.04 deg; joints [-10.812, -82.215, 118.211, -39.101, -31.419, 22.519] of KR 8 1620 ARC HW
    - target stk_p0_s5_t18 (Cartesian target) at (984.11, 169.3, 1037.38) mm, rotated rx 138.26 ry 76.5 rz 128.39 deg; joints [-11.531, -82.047, 118.008, -40.89, -31.971, 23.474] of KR 8 1620 ARC HW
    - target stk_p0_s5_t19 (Cartesian target) at (984.33, 179.86, 1037.51) mm, rotated rx 137.07 ry 76.25 rz 126.78 deg; joints [-12.245, -81.869, 117.793, -42.621, -32.541, 24.375] of KR 8 1620 ARC HW
    - target stk_p0_s5_t20 (Cartesian target) at (984.55, 190.42, 1037.63) mm, rotated rx 135.93 ry 75.99 rz 125.22 deg; joints [-12.954, -81.682, 117.566, -44.296, -33.126, 25.222] of KR 8 1620 ARC HW
    - target stk_p0_s5_t21 (Cartesian target) at (984.77, 200.98, 1037.76) mm, rotated rx 134.83 ry 75.72 rz 123.7 deg; joints [-13.659, -81.484, 117.327, -45.916, -33.726, 26.017] of KR 8 1620 ARC HW
    - target stk_p0_s5_t22 (Cartesian target) at (984.99, 211.54, 1037.88) mm, rotated rx 133.77 ry 75.45 rz 122.22 deg; joints [-14.359, -81.278, 117.076, -47.483, -34.34, 26.763] of KR 8 1620 ARC HW
    - target stk_p0_s5_t23 (Cartesian target) at (985.21, 222.09, 1038) mm, rotated rx 132.75 ry 75.18 rz 120.79 deg; joints [-15.054, -81.061, 116.812, -48.999, -34.965, 27.461] of KR 8 1620 ARC HW
    - target stk_p0_s5_t24 (Cartesian target) at (985.43, 232.65, 1038.13) mm, rotated rx 131.77 ry 74.9 rz 119.4 deg; joints [-15.744, -80.836, 116.536, -50.465, -35.601, 28.113] of KR 8 1620 ARC HW
    - target stk_p0_s5_t25 (Cartesian target) at (985.65, 243.21, 1038.25) mm, rotated rx 130.83 ry 74.62 rz 118.04 deg; joints [-16.428, -80.602, 116.248, -51.883, -36.247, 28.721] of KR 8 1620 ARC HW
    - target stk_p0_s6_t0 (Cartesian target) at (973.59, -337.5, 1031.45) mm, rotated rx -135.8 ry 76.35 rz -125.37 deg; joints [23.096, -78.494, 113.943, 57.198, -39.311, -34.399] of KR 8 1620 ARC HW
    - target stk_p0_s6_t0 (Cartesian target) at (973.59, -337.5, 1031.45) mm, rotated rx -135.8 ry 76.35 rz -125.37 deg; joints [23.096, -78.494, 113.943, 57.198, -39.311, -34.399] of KR 8 1620 ARC HW
    - target stk_p0_s6_t1 (Cartesian target) at (973.81, -326.94, 1031.58) mm, rotated rx -136.99 ry 76.6 rz -126.97 deg; joints [22.458, -78.794, 114.312, 55.99, -38.646, -33.976] of KR 8 1620 ARC HW
    - target stk_p0_s6_t2 (Cartesian target) at (974.03, -316.39, 1031.7) mm, rotated rx -138.23 ry 76.85 rz -128.62 deg; joints [21.814, -79.085, 114.669, 54.743, -37.986, -33.519] of KR 8 1620 ARC HW
    - target stk_p0_s6_t3 (Cartesian target) at (974.24, -305.83, 1031.83) mm, rotated rx -139.52 ry 77.09 rz -130.32 deg; joints [21.164, -79.368, 115.014, 53.457, -37.331, -33.026] of KR 8 1620 ARC HW
    - target stk_p0_s6_t4 (Cartesian target) at (974.46, -295.27, 1031.95) mm, rotated rx -140.85 ry 77.32 rz -132.08 deg; joints [20.508, -79.643, 115.347, 52.129, -36.683, -32.497] of KR 8 1620 ARC HW
    - target stk_p0_s6_t5 (Cartesian target) at (974.68, -284.71, 1032.07) mm, rotated rx -142.24 ry 77.55 rz -133.88 deg; joints [19.845, -79.91, 115.668, 50.757, -36.042, -31.929] of KR 8 1620 ARC HW
    - target stk_p0_s6_t6 (Cartesian target) at (974.9, -274.15, 1032.2) mm, rotated rx -143.69 ry 77.77 rz -135.74 deg; joints [19.177, -80.168, 115.978, 49.341, -35.409, -31.319] of KR 8 1620 ARC HW
    - target stk_p0_s6_t7 (Cartesian target) at (975.12, -263.59, 1032.32) mm, rotated rx -145.18 ry 77.98 rz -137.65 deg; joints [18.503, -80.417, 116.275, 47.877, -34.786, -30.666] of KR 8 1620 ARC HW
    - target stk_p0_s6_t8 (Cartesian target) at (975.34, -253.04, 1032.44) mm, rotated rx -146.73 ry 78.19 rz -139.62 deg; joints [17.823, -80.658, 116.561, 46.363, -34.174, -29.968] of KR 8 1620 ARC HW
    - target stk_p0_s6_t9 (Cartesian target) at (975.56, -242.48, 1032.57) mm, rotated rx -148.34 ry 78.38 rz -141.65 deg; joints [17.138, -80.889, 116.834, 44.799, -33.573, -29.222] of KR 8 1620 ARC HW
    - target stk_p0_s6_t10 (Cartesian target) at (975.78, -231.92, 1032.69) mm, rotated rx -150 ry 78.57 rz -143.73 deg; joints [16.448, -81.112, 117.096, 43.183, -32.985, -28.428] of KR 8 1620 ARC HW
    - target stk_p0_s6_t11 (Cartesian target) at (976, -221.36, 1032.81) mm, rotated rx -151.72 ry 78.75 rz -145.87 deg; joints [15.752, -81.325, 117.345, 41.512, -32.411, -27.582] of KR 8 1620 ARC HW
    - target stk_p0_s6_t12 (Cartesian target) at (976.22, -210.8, 1032.94) mm, rotated rx -153.49 ry 78.92 rz -148.06 deg; joints [15.051, -81.529, 117.582, 39.784, -31.852, -26.683] of KR 8 1620 ARC HW
    - target stk_p0_s6_t13 (Cartesian target) at (976.44, -200.24, 1033.06) mm, rotated rx -155.32 ry 79.07 rz -150.32 deg; joints [14.346, -81.724, 117.808, 38, -31.311, -25.73] of KR 8 1620 ARC HW
    - target stk_p0_s6_t14 (Cartesian target) at (976.66, -189.68, 1033.18) mm, rotated rx -157.21 ry 79.22 rz -152.62 deg; joints [13.636, -81.909, 118.021, 36.157, -30.789, -24.721] of KR 8 1620 ARC HW
    - target stk_p0_s6_t15 (Cartesian target) at (976.88, -179.13, 1033.31) mm, rotated rx -159.14 ry 79.36 rz -154.98 deg; joints [12.921, -82.084, 118.222, 34.255, -30.286, -23.655] of KR 8 1620 ARC HW
    - target stk_p0_s6_t16 (Cartesian target) at (977.1, -168.57, 1033.43) mm, rotated rx -161.12 ry 79.48 rz -157.39 deg; joints [12.202, -82.25, 118.411, 32.293, -29.805, -22.532] of KR 8 1620 ARC HW
    - target stk_p0_s6_t17 (Cartesian target) at (977.31, -158.01, 1033.55) mm, rotated rx -163.15 ry 79.59 rz -159.84 deg; joints [11.479, -82.405, 118.588, 30.271, -29.348, -21.351] of KR 8 1620 ARC HW
    - target stk_p0_s6_t18 (Cartesian target) at (977.53, -147.45, 1033.68) mm, rotated rx -165.23 ry 79.69 rz -162.34 deg; joints [10.753, -82.551, 118.753, 28.189, -28.916, -20.113] of KR 8 1620 ARC HW
    - target stk_p0_s6_t19 (Cartesian target) at (977.75, -136.89, 1033.8) mm, rotated rx -167.34 ry 79.77 rz -164.87 deg; joints [10.022, -82.687, 118.906, 26.048, -28.51, -18.817] of KR 8 1620 ARC HW
    - target stk_p0_s6_t20 (Cartesian target) at (977.97, -126.33, 1033.93) mm, rotated rx -169.48 ry 79.84 rz -167.44 deg; joints [9.289, -82.813, 119.046, 23.85, -28.133, -17.466] of KR 8 1620 ARC HW
    - target stk_p0_s6_t21 (Cartesian target) at (978.19, -115.78, 1034.05) mm, rotated rx -171.65 ry 79.9 rz -170.04 deg; joints [8.552, -82.928, 119.175, 21.596, -27.786, -16.061] of KR 8 1620 ARC HW
    - target stk_p0_s6_t22 (Cartesian target) at (978.41, -105.22, 1034.17) mm, rotated rx -173.85 ry 79.94 rz -172.66 deg; joints [7.812, -83.033, 119.291, 19.29, -27.47, -14.604] of KR 8 1620 ARC HW
    - target stk_p0_s6_t23 (Cartesian target) at (978.63, -94.66, 1034.3) mm, rotated rx -176.06 ry 79.97 rz -175.3 deg; joints [7.07, -83.128, 119.395, 16.934, -27.188, -13.099] of KR 8 1620 ARC HW
    - target stk_p0_s6_t24 (Cartesian target) at (978.85, -84.1, 1034.42) mm, rotated rx -178.28 ry 79.98 rz -177.95 deg; joints [6.325, -83.212, 119.487, 14.532, -26.94, -11.55] of KR 8 1620 ARC HW
    - target stk_p0_s6_t25 (Cartesian target) at (979.07, -73.54, 1034.54) mm, rotated rx 179.5 ry 79.98 rz 179.4 deg; joints [5.579, -83.286, 119.566, 12.091, -26.728, -9.962] of KR 8 1620 ARC HW
    - target stk_p1_s7_t0 (Cartesian target) at (979.76, -18.02, 802.83) mm, rotated rx 124.86 ry 87.37 rz 122.67 deg; joints [1.941, -74.976, 132.377, -0.258, -55.901, -2.016] of KR 8 1620 ARC HW
    - target stk_p1_s7_t0 (Cartesian target) at (979.76, -18.02, 802.83) mm, rotated rx 124.86 ry 87.37 rz 122.67 deg; joints [1.941, -74.976, 132.377, -0.258, -55.901, -2.016] of KR 8 1620 ARC HW
    - target stk_p1_s7_t1 (Cartesian target) at (979.98, -7.46, 802.95) mm, rotated rx 120.58 ry 87.04 rz 118 deg; joints [1.195, -74.987, 132.39, -1.633, -55.909, -1.668] of KR 8 1620 ARC HW
    - target stk_p1_s7_t2 (Cartesian target) at (980.2, 3.09, 803.07) mm, rotated rx 117.18 ry 86.7 rz 114.2 deg; joints [0.448, -74.989, 132.39, -3.008, -55.927, -1.32] of KR 8 1620 ARC HW
    - target stk_p1_s7_t3 (Cartesian target) at (980.42, 13.65, 803.2) mm, rotated rx 114.43 ry 86.34 rz 111.06 deg; joints [-0.298, -74.982, 132.378, -4.382, -55.957, -0.972] of KR 8 1620 ARC HW
    - target stk_p1_s7_t4 (Cartesian target) at (980.64, 24.21, 803.32) mm, rotated rx 112.18 ry 85.98 rz 108.4 deg; joints [-1.044, -74.966, 132.352, -5.754, -55.998, -0.626] of KR 8 1620 ARC HW
    - target stk_p1_s7_t5 (Cartesian target) at (980.86, 34.77, 803.44) mm, rotated rx 110.3 ry 85.61 rz 106.13 deg; joints [-1.79, -74.941, 132.314, -7.124, -56.049, -0.281] of KR 8 1620 ARC HW
    - target stk_p1_s7_t6 (Cartesian target) at (981.08, 45.33, 803.57) mm, rotated rx 108.71 ry 85.24 rz 104.14 deg; joints [-2.535, -74.907, 132.263, -8.492, -56.112, 0.062] of KR 8 1620 ARC HW
    - target stk_p1_s7_t7 (Cartesian target) at (981.3, 55.89, 803.69) mm, rotated rx 107.35 ry 84.87 rz 102.39 deg; joints [-3.279, -74.864, 132.199, -9.856, -56.185, 0.402] of KR 8 1620 ARC HW
    - target stk_p1_s7_t8 (Cartesian target) at (981.52, 66.44, 803.81) mm, rotated rx 106.18 ry 84.49 rz 100.82 deg; joints [-4.021, -74.811, 132.122, -11.216, -56.269, 0.741] of KR 8 1620 ARC HW
    - target stk_p1_s7_t9 (Cartesian target) at (981.73, 77, 803.94) mm, rotated rx 105.16 ry 84.11 rz 99.4 deg; joints [-4.762, -74.75, 132.032, -12.571, -56.364, 1.076] of KR 8 1620 ARC HW
    - target stk_p1_s7_t10 (Cartesian target) at (981.95, 87.56, 804.06) mm, rotated rx 104.26 ry 83.74 rz 98.11 deg; joints [-5.5, -74.679, 131.93, -13.921, -56.469, 1.408] of KR 8 1620 ARC HW
    - target stk_p1_s7_t11 (Cartesian target) at (982.17, 98.12, 804.18) mm, rotated rx 103.47 ry 83.36 rz 96.92 deg; joints [-6.237, -74.6, 131.814, -15.264, -56.584, 1.737] of KR 8 1620 ARC HW
    - target stk_p1_s7_t12 (Cartesian target) at (982.39, 108.68, 804.31) mm, rotated rx 102.76 ry 82.98 rz 95.82 deg; joints [-6.971, -74.512, 131.686, -16.602, -56.709, 2.062] of KR 8 1620 ARC HW
    - target stk_p1_s7_t13 (Cartesian target) at (982.61, 119.24, 804.43) mm, rotated rx 102.13 ry 82.6 rz 94.79 deg; joints [-7.703, -74.415, 131.545, -17.932, -56.844, 2.383] of KR 8 1620 ARC HW
    - target stk_p1_s7_t14 (Cartesian target) at (982.83, 129.79, 804.56) mm, rotated rx 101.55 ry 82.22 rz 93.82 deg; joints [-8.431, -74.309, 131.391, -19.255, -56.989, 2.699] of KR 8 1620 ARC HW
    - target stk_p1_s7_t15 (Cartesian target) at (983.05, 140.35, 804.68) mm, rotated rx 101.04 ry 81.83 rz 92.91 deg; joints [-9.157, -74.195, 131.225, -20.57, -57.143, 3.011] of KR 8 1620 ARC HW
    - target stk_p1_s7_t16 (Cartesian target) at (983.27, 150.91, 804.8) mm, rotated rx 100.56 ry 81.45 rz 92.05 deg; joints [-9.879, -74.071, 131.046, -21.877, -57.306, 3.318] of KR 8 1620 ARC HW
    - target stk_p1_s7_t17 (Cartesian target) at (983.49, 161.47, 804.93) mm, rotated rx 100.13 ry 81.07 rz 91.22 deg; joints [-10.597, -73.94, 130.854, -23.174, -57.478, 3.62] of KR 8 1620 ARC HW
    - target stk_p1_s7_t18 (Cartesian target) at (983.71, 172.03, 805.05) mm, rotated rx 99.74 ry 80.69 rz 90.44 deg; joints [-11.312, -73.8, 130.65, -24.463, -57.659, 3.917] of KR 8 1620 ARC HW
    - target stk_p1_s7_t19 (Cartesian target) at (983.93, 182.59, 805.17) mm, rotated rx 99.37 ry 80.31 rz 89.68 deg; joints [-12.022, -73.651, 130.433, -25.741, -57.849, 4.209] of KR 8 1620 ARC HW
    - target stk_p1_s7_t20 (Cartesian target) at (984.15, 193.15, 805.3) mm, rotated rx 99.04 ry 79.93 rz 88.96 deg; joints [-12.728, -73.494, 130.204, -27.01, -58.047, 4.495] of KR 8 1620 ARC HW
    - target stk_p1_s7_t21 (Cartesian target) at (984.37, 203.7, 805.42) mm, rotated rx 98.73 ry 79.55 rz 88.26 deg; joints [-13.43, -73.329, 129.962, -28.268, -58.253, 4.776] of KR 8 1620 ARC HW
    - target stk_p1_s7_t22 (Cartesian target) at (984.59, 214.26, 805.54) mm, rotated rx 98.44 ry 79.17 rz 87.58 deg; joints [-14.128, -73.156, 129.708, -29.515, -58.466, 5.051] of KR 8 1620 ARC HW
    - target stk_p1_s7_t23 (Cartesian target) at (984.81, 224.82, 805.67) mm, rotated rx 98.17 ry 78.8 rz 86.92 deg; joints [-14.82, -72.975, 129.441, -30.751, -58.687, 5.321] of KR 8 1620 ARC HW
    - target stk_p1_s7_t24 (Cartesian target) at (985.02, 235.38, 805.79) mm, rotated rx 97.92 ry 78.42 rz 86.29 deg; joints [-15.508, -72.786, 129.162, -31.976, -58.915, 5.586] of KR 8 1620 ARC HW
    - target stk_p1_s7_t25 (Cartesian target) at (985.24, 245.94, 805.91) mm, rotated rx 97.68 ry 78.04 rz 85.66 deg; joints [-16.19, -72.589, 128.871, -33.19, -59.15, 5.844] of KR 8 1620 ARC HW
    - target stk_p1_s8_t0 (Cartesian target) at (973.18, -334.78, 799.12) mm, rotated rx -98.05 ry 80.4 rz -88.43 deg; joints [23.017, -70.646, 126.139, 38.267, -60.213, -11.038] of KR 8 1620 ARC HW
    - target stk_p1_s8_t0 (Cartesian target) at (973.18, -334.78, 799.12) mm, rotated rx -98.05 ry 80.4 rz -88.43 deg; joints [23.017, -70.646, 126.139, 38.267, -60.213, -11.038] of KR 8 1620 ARC HW
    - target stk_p1_s8_t1 (Cartesian target) at (973.4, -324.22, 799.24) mm, rotated rx -98.42 ry 80.78 rz -89.18 deg; joints [22.384, -70.902, 126.522, 37.129, -59.957, -10.807] of KR 8 1620 ARC HW
    - target stk_p1_s8_t2 (Cartesian target) at (973.62, -313.66, 799.37) mm, rotated rx -98.82 ry 81.15 rz -89.97 deg; joints [21.744, -71.152, 126.894, 35.978, -59.707, -10.57] of KR 8 1620 ARC HW
    - target stk_p1_s8_t3 (Cartesian target) at (973.84, -303.1, 799.49) mm, rotated rx -99.25 ry 81.53 rz -90.79 deg; joints [21.099, -71.395, 127.254, 34.815, -59.463, -10.329] of KR 8 1620 ARC HW
    - target stk_p1_s8_t4 (Cartesian target) at (974.06, -292.54, 799.61) mm, rotated rx -99.72 ry 81.9 rz -91.65 deg; joints [20.448, -71.631, 127.603, 33.64, -59.224, -10.082] of KR 8 1620 ARC HW
    - target stk_p1_s8_t5 (Cartesian target) at (974.28, -281.98, 799.74) mm, rotated rx -100.24 ry 82.28 rz -92.56 deg; joints [19.791, -71.859, 127.94, 32.452, -58.992, -9.83] of KR 8 1620 ARC HW
    - target stk_p1_s8_t6 (Cartesian target) at (974.5, -271.43, 799.86) mm, rotated rx -100.82 ry 82.66 rz -93.52 deg; joints [19.128, -72.081, 128.265, 31.253, -58.766, -9.573] of KR 8 1620 ARC HW
    - target stk_p1_s8_t7 (Cartesian target) at (974.72, -260.87, 799.98) mm, rotated rx -101.46 ry 83.03 rz -94.55 deg; joints [18.46, -72.295, 128.578, 30.042, -58.547, -9.31] of KR 8 1620 ARC HW
    - target stk_p1_s8_t8 (Cartesian target) at (974.94, -250.31, 800.11) mm, rotated rx -102.17 ry 83.41 rz -95.65 deg; joints [17.787, -72.502, 128.879, 28.82, -58.335, -9.042] of KR 8 1620 ARC HW
    - target stk_p1_s8_t9 (Cartesian target) at (975.16, -239.75, 800.23) mm, rotated rx -102.97 ry 83.78 rz -96.84 deg; joints [17.108, -72.701, 129.168, 27.586, -58.13, -8.768] of KR 8 1620 ARC HW
    - target stk_p1_s8_t10 (Cartesian target) at (975.37, -229.19, 800.35) mm, rotated rx -103.88 ry 84.16 rz -98.14 deg; joints [16.423, -72.893, 129.445, 26.341, -57.933, -8.49] of KR 8 1620 ARC HW
    - target stk_p1_s8_t11 (Cartesian target) at (975.59, -218.63, 800.48) mm, rotated rx -104.9 ry 84.53 rz -99.56 deg; joints [15.734, -73.077, 129.71, 25.086, -57.743, -8.206] of KR 8 1620 ARC HW
    - target stk_p1_s8_t12 (Cartesian target) at (975.81, -208.07, 800.6) mm, rotated rx -106.09 ry 84.91 rz -101.13 deg; joints [15.04, -73.252, 129.963, 23.82, -57.562, -7.916] of KR 8 1620 ARC HW
    - target stk_p1_s8_t13 (Cartesian target) at (976.03, -197.52, 800.73) mm, rotated rx -107.45 ry 85.28 rz -102.89 deg; joints [14.341, -73.42, 130.203, 22.544, -57.388, -7.622] of KR 8 1620 ARC HW
    - target stk_p1_s8_t14 (Cartesian target) at (976.25, -186.96, 800.85) mm, rotated rx -109.06 ry 85.65 rz -104.89 deg; joints [13.638, -73.58, 130.431, 21.258, -57.223, -7.322] of KR 8 1620 ARC HW
    - target stk_p1_s8_t15 (Cartesian target) at (976.47, -176.4, 800.97) mm, rotated rx -110.96 ry 86.01 rz -107.18 deg; joints [12.93, -73.732, 130.647, 19.963, -57.066, -7.018] of KR 8 1620 ARC HW
    - target stk_p1_s8_t16 (Cartesian target) at (976.69, -165.84, 801.1) mm, rotated rx -113.23 ry 86.37 rz -109.86 deg; joints [12.218, -73.876, 130.851, 18.659, -56.919, -6.708] of KR 8 1620 ARC HW
    - target stk_p1_s8_t17 (Cartesian target) at (976.91, -155.28, 801.22) mm, rotated rx -116.01 ry 86.72 rz -113.03 deg; joints [11.502, -74.011, 131.042, 17.347, -56.781, -6.395] of KR 8 1620 ARC HW
    - target stk_p1_s8_t18 (Cartesian target) at (977.13, -144.72, 801.34) mm, rotated rx -119.45 ry 87.07 rz -116.87 deg; joints [10.783, -74.138, 131.22, 16.026, -56.652, -6.076] of KR 8 1620 ARC HW
    - target stk_p1_s8_t19 (Cartesian target) at (977.35, -134.17, 801.47) mm, rotated rx -123.79 ry 87.4 rz -121.6 deg; joints [10.06, -74.256, 131.387, 14.698, -56.532, -5.754] of KR 8 1620 ARC HW
    - target stk_p1_s8_t20 (Cartesian target) at (977.57, -123.61, 801.59) mm, rotated rx -129.35 ry 87.71 rz -127.56 deg; joints [9.334, -74.366, 131.54, 13.363, -56.423, -5.428] of KR 8 1620 ARC HW
    - target stk_p1_s8_t21 (Cartesian target) at (977.79, -113.05, 801.71) mm, rotated rx -136.58 ry 87.99 rz -135.18 deg; joints [8.604, -74.467, 131.681, 12.021, -56.323, -5.098] of KR 8 1620 ARC HW
    - target stk_p1_s8_t22 (Cartesian target) at (978.01, -102.49, 801.84) mm, rotated rx -145.98 ry 88.24 rz -144.98 deg; joints [7.872, -74.559, 131.809, 10.673, -56.234, -4.764] of KR 8 1620 ARC HW
    - target stk_p1_s8_t23 (Cartesian target) at (978.23, -91.93, 801.96) mm, rotated rx -157.93 ry 88.42 rz -157.33 deg; joints [7.137, -74.642, 131.925, 9.319, -56.155, -4.428] of KR 8 1620 ARC HW
    - target stk_p1_s8_t24 (Cartesian target) at (978.45, -81.37, 802.08) mm, rotated rx -172.17 ry 88.51 rz -171.97 deg; joints [6.4, -74.717, 132.028, 7.961, -56.086, -4.089] of KR 8 1620 ARC HW
    - target stk_p1_s8_t25 (Cartesian target) at (978.66, -70.82, 802.21) mm, rotated rx 172.66 ry 88.51 rz 172.47 deg; joints [5.66, -74.783, 132.118, 6.598, -56.028, -3.747] of KR 8 1620 ARC HW
    - target stk_p1_s9_t0 (Cartesian target) at (979.95, -19.26, 908.43) mm, rotated rx 158.78 ry 84.19 rz 156.57 deg; joints [2.029, -79.825, 126.86, -0.12, -41.622, -2.026] of KR 8 1620 ARC HW
    - target stk_p1_s9_t0 (Cartesian target) at (979.95, -19.26, 908.43) mm, rotated rx 158.78 ry 84.19 rz 156.57 deg; joints [2.029, -79.825, 126.86, -0.12, -41.622, -2.026] of KR 8 1620 ARC HW
    - target stk_p1_s9_t1 (Cartesian target) at (980.16, -8.7, 908.56) mm, rotated rx 155.29 ry 84.03 rz 152.66 deg; joints [1.283, -79.838, 126.874, -1.826, -41.632, -1.252] of KR 8 1620 ARC HW
    - target stk_p1_s9_t2 (Cartesian target) at (980.38, 1.85, 908.68) mm, rotated rx 151.98 ry 83.86 rz 148.95 deg; joints [0.538, -79.842, 126.876, -3.531, -41.663, -0.478] of KR 8 1620 ARC HW
    - target stk_p1_s9_t3 (Cartesian target) at (980.6, 12.41, 908.8) mm, rotated rx 148.88 ry 83.66 rz 145.43 deg; joints [-0.208, -79.835, 126.866, -5.233, -41.715, 0.293] of KR 8 1620 ARC HW
    - target stk_p1_s9_t4 (Cartesian target) at (980.82, 22.97, 908.93) mm, rotated rx 145.96 ry 83.45 rz 142.11 deg; joints [-0.953, -79.819, 126.844, -6.93, -41.788, 1.06] of KR 8 1620 ARC HW
    - target stk_p1_s9_t5 (Cartesian target) at (981.04, 33.53, 909.05) mm, rotated rx 143.24 ry 83.22 rz 138.98 deg; joints [-1.698, -79.793, 126.809, -8.621, -41.881, 1.821] of KR 8 1620 ARC HW
    - target stk_p1_s9_t6 (Cartesian target) at (981.26, 44.09, 909.17) mm, rotated rx 140.71 ry 82.97 rz 136.03 deg; joints [-2.442, -79.757, 126.761, -10.305, -41.995, 2.575] of KR 8 1620 ARC HW
    - target stk_p1_s9_t7 (Cartesian target) at (981.48, 54.65, 909.3) mm, rotated rx 138.35 ry 82.72 rz 133.26 deg; joints [-3.185, -79.711, 126.702, -11.979, -42.129, 3.321] of KR 8 1620 ARC HW
    - target stk_p1_s9_t8 (Cartesian target) at (981.7, 65.2, 909.42) mm, rotated rx 136.15 ry 82.45 rz 130.66 deg; joints [-3.926, -79.655, 126.63, -13.643, -42.283, 4.057] of KR 8 1620 ARC HW
    - target stk_p1_s9_t9 (Cartesian target) at (981.92, 75.76, 909.54) mm, rotated rx 134.11 ry 82.17 rz 128.2 deg; joints [-4.666, -79.589, 126.545, -15.294, -42.456, 4.783] of KR 8 1620 ARC HW
    - target stk_p1_s9_t10 (Cartesian target) at (982.14, 86.32, 909.67) mm, rotated rx 132.21 ry 81.89 rz 125.9 deg; joints [-5.404, -79.514, 126.449, -16.932, -42.648, 5.496] of KR 8 1620 ARC HW
    - target stk_p1_s9_t11 (Cartesian target) at (982.36, 96.88, 909.79) mm, rotated rx 130.44 ry 81.59 rz 123.72 deg; joints [-6.14, -79.428, 126.34, -18.555, -42.858, 6.196] of KR 8 1620 ARC HW
    - target stk_p1_s9_t12 (Cartesian target) at (982.58, 107.44, 909.92) mm, rotated rx 128.8 ry 81.29 rz 121.67 deg; joints [-6.874, -79.333, 126.218, -20.162, -43.086, 6.881] of KR 8 1620 ARC HW
    - target stk_p1_s9_t13 (Cartesian target) at (982.8, 118, 910.04) mm, rotated rx 127.26 ry 80.99 rz 119.73 deg; joints [-7.605, -79.229, 126.085, -21.752, -43.332, 7.552] of KR 8 1620 ARC HW
    - target stk_p1_s9_t14 (Cartesian target) at (983.02, 128.56, 910.16) mm, rotated rx 125.83 ry 80.67 rz 117.89 deg; joints [-8.333, -79.115, 125.939, -23.324, -43.595, 8.207] of KR 8 1620 ARC HW
    - target stk_p1_s9_t15 (Cartesian target) at (983.23, 139.11, 910.29) mm, rotated rx 124.5 ry 80.36 rz 116.15 deg; joints [-9.058, -78.991, 125.78, -24.877, -43.874, 8.846] of KR 8 1620 ARC HW
    - target stk_p1_s9_t16 (Cartesian target) at (983.45, 149.67, 910.41) mm, rotated rx 123.25 ry 80.03 rz 114.49 deg; joints [-9.78, -78.858, 125.61, -26.41, -44.169, 9.467] of KR 8 1620 ARC HW
    - target stk_p1_s9_t17 (Cartesian target) at (983.67, 160.23, 910.53) mm, rotated rx 122.08 ry 79.71 rz 112.92 deg; joints [-10.498, -78.716, 125.427, -27.923, -44.479, 10.071] of KR 8 1620 ARC HW
    - target stk_p1_s9_t18 (Cartesian target) at (983.89, 170.79, 910.66) mm, rotated rx 120.99 ry 79.38 rz 111.42 deg; joints [-11.213, -78.564, 125.232, -29.415, -44.803, 10.657] of KR 8 1620 ARC HW
    - target stk_p1_s9_t19 (Cartesian target) at (984.11, 181.35, 910.78) mm, rotated rx 119.96 ry 79.05 rz 109.99 deg; joints [-11.923, -78.404, 125.025, -30.886, -45.142, 11.225] of KR 8 1620 ARC HW
    - target stk_p1_s9_t20 (Cartesian target) at (984.33, 191.91, 910.9) mm, rotated rx 118.99 ry 78.71 rz 108.62 deg; joints [-12.629, -78.234, 124.806, -32.334, -45.493, 11.775] of KR 8 1620 ARC HW
    - target stk_p1_s9_t21 (Cartesian target) at (984.55, 202.46, 911.03) mm, rotated rx 118.08 ry 78.38 rz 107.31 deg; joints [-13.331, -78.055, 124.574, -33.761, -45.857, 12.306] of KR 8 1620 ARC HW
    - target stk_p1_s9_t22 (Cartesian target) at (984.77, 213.02, 911.15) mm, rotated rx 117.22 ry 78.04 rz 106.05 deg; joints [-14.029, -77.868, 124.331, -35.166, -46.233, 12.818] of KR 8 1620 ARC HW
    - target stk_p1_s9_t23 (Cartesian target) at (984.99, 223.58, 911.27) mm, rotated rx 116.42 ry 77.7 rz 104.84 deg; joints [-14.721, -77.672, 124.075, -36.547, -46.62, 13.312] of KR 8 1620 ARC HW
    - target stk_p1_s9_t24 (Cartesian target) at (985.21, 234.14, 911.4) mm, rotated rx 115.65 ry 77.36 rz 103.68 deg; joints [-15.409, -77.467, 123.807, -37.907, -47.017, 13.788] of KR 8 1620 ARC HW
    - target stk_p1_s9_t25 (Cartesian target) at (985.43, 244.7, 911.52) mm, rotated rx 114.93 ry 77.02 rz 102.56 deg; joints [-16.091, -77.254, 123.527, -39.243, -47.425, 14.246] of KR 8 1620 ARC HW
    - target stk_p1_s10_t0 (Cartesian target) at (973.37, -336.02, 904.73) mm, rotated rx -118.67 ry 79.14 rz -108.69 deg; joints [23.057, -75.085, 120.789, 44.967, -49.416, -20.154] of KR 8 1620 ARC HW
    - target stk_p1_s10_t0 (Cartesian target) at (973.37, -336.02, 904.73) mm, rotated rx -118.67 ry 79.14 rz -108.69 deg; joints [23.057, -75.085, 120.789, 44.967, -49.416, -20.154] of KR 8 1620 ARC HW
    - target stk_p1_s10_t1 (Cartesian target) at (973.59, -325.46, 904.85) mm, rotated rx -119.7 ry 79.47 rz -110.11 deg; joints [22.426, -75.365, 121.163, 43.758, -48.981, -19.785] of KR 8 1620 ARC HW
    - target stk_p1_s10_t2 (Cartesian target) at (973.8, -314.9, 904.97) mm, rotated rx -120.8 ry 79.79 rz -111.61 deg; joints [21.788, -75.637, 121.525, 42.526, -48.552, -19.4] of KR 8 1620 ARC HW
    - target stk_p1_s10_t3 (Cartesian target) at (974.02, -304.34, 905.1) mm, rotated rx -121.98 ry 80.11 rz -113.18 deg; joints [21.144, -75.902, 121.876, 41.273, -48.131, -18.999] of KR 8 1620 ARC HW
    - target stk_p1_s10_t4 (Cartesian target) at (974.24, -293.78, 905.22) mm, rotated rx -123.23 ry 80.43 rz -114.84 deg; joints [20.495, -76.159, 122.215, 39.997, -47.717, -18.581] of KR 8 1620 ARC HW
    - target stk_p1_s10_t5 (Cartesian target) at (974.46, -283.22, 905.34) mm, rotated rx -124.57 ry 80.74 rz -116.58 deg; joints [19.84, -76.408, 122.543, 38.7, -47.312, -18.146] of KR 8 1620 ARC HW
    - target stk_p1_s10_t6 (Cartesian target) at (974.68, -272.66, 905.47) mm, rotated rx -126.01 ry 81.05 rz -118.41 deg; joints [19.179, -76.65, 122.859, 37.38, -46.915, -17.694] of KR 8 1620 ARC HW
    - target stk_p1_s10_t7 (Cartesian target) at (974.9, -262.11, 905.59) mm, rotated rx -127.55 ry 81.35 rz -120.35 deg; joints [18.512, -76.884, 123.163, 36.037, -46.528, -17.224] of KR 8 1620 ARC HW
    - target stk_p1_s10_t8 (Cartesian target) at (975.12, -251.55, 905.71) mm, rotated rx -129.2 ry 81.65 rz -122.41 deg; joints [17.84, -77.11, 123.455, 34.672, -46.152, -16.736] of KR 8 1620 ARC HW
    - target stk_p1_s10_t9 (Cartesian target) at (975.34, -240.99, 905.84) mm, rotated rx -130.97 ry 81.94 rz -124.59 deg; joints [17.163, -77.327, 123.736, 33.285, -45.785, -16.23] of KR 8 1620 ARC HW
    - target stk_p1_s10_t10 (Cartesian target) at (975.56, -230.43, 905.96) mm, rotated rx -132.88 ry 82.22 rz -126.9 deg; joints [16.48, -77.536, 124.005, 31.875, -45.431, -15.706] of KR 8 1620 ARC HW
    - target stk_p1_s10_t11 (Cartesian target) at (975.78, -219.87, 906.09) mm, rotated rx -134.93 ry 82.49 rz -129.35 deg; joints [15.793, -77.737, 124.262, 30.443, -45.088, -15.164] of KR 8 1620 ARC HW
    - target stk_p1_s10_t12 (Cartesian target) at (976, -209.31, 906.21) mm, rotated rx -137.13 ry 82.76 rz -131.96 deg; joints [15.1, -77.93, 124.508, 28.989, -44.757, -14.604] of KR 8 1620 ARC HW
    - target stk_p1_s10_t13 (Cartesian target) at (976.22, -198.76, 906.33) mm, rotated rx -139.51 ry 83.01 rz -134.74 deg; joints [14.403, -78.113, 124.741, 27.513, -44.44, -14.026] of KR 8 1620 ARC HW
    - target stk_p1_s10_t14 (Cartesian target) at (976.44, -188.2, 906.46) mm, rotated rx -142.05 ry 83.25 rz -137.69 deg; joints [13.702, -78.288, 124.962, 26.017, -44.137, -13.431] of KR 8 1620 ARC HW
    - target stk_p1_s10_t15 (Cartesian target) at (976.66, -177.64, 906.58) mm, rotated rx -144.78 ry 83.48 rz -140.83 deg; joints [12.996, -78.455, 125.172, 24.499, -43.848, -12.818] of KR 8 1620 ARC HW
    - target stk_p1_s10_t16 (Cartesian target) at (976.87, -167.08, 906.7) mm, rotated rx -147.7 ry 83.69 rz -144.16 deg; joints [12.285, -78.612, 125.37, 22.961, -43.574, -12.187] of KR 8 1620 ARC HW
    - target stk_p1_s10_t17 (Cartesian target) at (977.09, -156.52, 906.83) mm, rotated rx -150.82 ry 83.88 rz -147.69 deg; joints [11.571, -78.76, 125.555, 21.404, -43.316, -11.541] of KR 8 1620 ARC HW
    - target stk_p1_s10_t18 (Cartesian target) at (977.31, -145.96, 906.95) mm, rotated rx -154.14 ry 84.05 rz -151.41 deg; joints [10.853, -78.899, 125.728, 19.829, -43.074, -10.878] of KR 8 1620 ARC HW
    - target stk_p1_s10_t19 (Cartesian target) at (977.53, -135.41, 907.07) mm, rotated rx -157.64 ry 84.21 rz -155.33 deg; joints [10.132, -79.029, 125.89, 18.235, -42.849, -10.2] of KR 8 1620 ARC HW
    - target stk_p1_s10_t20 (Cartesian target) at (977.75, -124.85, 907.2) mm, rotated rx -161.32 ry 84.34 rz -159.42 deg; joints [9.407, -79.149, 126.039, 16.625, -42.641, -9.508] of KR 8 1620 ARC HW
    - target stk_p1_s10_t21 (Cartesian target) at (977.97, -114.29, 907.32) mm, rotated rx -165.17 ry 84.45 rz -163.67 deg; joints [8.679, -79.26, 126.176, 14.999, -42.452, -8.802] of KR 8 1620 ARC HW
    - target stk_p1_s10_t22 (Cartesian target) at (978.19, -103.73, 907.44) mm, rotated rx -169.14 ry 84.53 rz -168.06 deg; joints [7.948, -79.362, 126.301, 13.359, -42.28, -8.083] of KR 8 1620 ARC HW
    - target stk_p1_s10_t23 (Cartesian target) at (978.41, -93.17, 907.57) mm, rotated rx -173.22 ry 84.58 rz -172.55 deg; joints [7.215, -79.454, 126.414, 11.705, -42.128, -7.353] of KR 8 1620 ARC HW
    - target stk_p1_s10_t24 (Cartesian target) at (978.63, -82.61, 907.69) mm, rotated rx -177.36 ry 84.61 rz -177.1 deg; joints [6.479, -79.536, 126.514, 10.039, -41.995, -6.612] of KR 8 1620 ARC HW
    - target stk_p1_s10_t25 (Cartesian target) at (978.85, -72.05, 907.81) mm, rotated rx 178.47 ry 84.61 rz 178.32 deg; joints [5.741, -79.609, 126.603, 8.363, -41.882, -5.863] of KR 8 1620 ARC HW
    - target stk_p1_s11_t0 (Cartesian target) at (973, -333.54, 693.51) mm, rotated rx -75.01 ry 80.21 rz -65.76 deg; joints [22.96, -64.898, 130.134, 34.334, -71.741, -4.218] of KR 8 1620 ARC HW
    - target stk_p1_s11_t0 (Cartesian target) at (973, -333.54, 693.51) mm, rotated rx -75.01 ry 80.21 rz -65.76 deg; joints [22.96, -64.898, 130.134, 34.334, -71.741, -4.218] of KR 8 1620 ARC HW
    - target stk_p1_s11_t1 (Cartesian target) at (973.22, -322.98, 693.64) mm, rotated rx -74.43 ry 80.58 rz -65.54 deg; joints [22.325, -65.122, 130.527, 33.265, -71.644, -4.128] of KR 8 1620 ARC HW
    - target stk_p1_s11_t2 (Cartesian target) at (973.44, -312.42, 693.76) mm, rotated rx -73.79 ry 80.95 rz -65.28 deg; joints [21.685, -65.34, 130.908, 32.188, -71.551, -4.041] of KR 8 1620 ARC HW
    - target stk_p1_s11_t3 (Cartesian target) at (973.66, -301.86, 693.88) mm, rotated rx -73.11 ry 81.31 rz -64.97 deg; joints [21.038, -65.552, 131.277, 31.103, -71.461, -3.955] of KR 8 1620 ARC HW
    - target stk_p1_s11_t4 (Cartesian target) at (973.87, -291.3, 694.01) mm, rotated rx -72.36 ry 81.68 rz -64.6 deg; joints [20.386, -65.757, 131.634, 30.011, -71.374, -3.87] of KR 8 1620 ARC HW
    - target stk_p1_s11_t5 (Cartesian target) at (974.09, -280.74, 694.13) mm, rotated rx -71.54 ry 82.04 rz -64.15 deg; joints [19.728, -65.956, 131.98, 28.911, -71.291, -3.788] of KR 8 1620 ARC HW
    - target stk_p1_s11_t6 (Cartesian target) at (974.31, -270.19, 694.25) mm, rotated rx -70.64 ry 82.41 rz -63.63 deg; joints [19.064, -66.149, 132.313, 27.804, -71.211, -3.707] of KR 8 1620 ARC HW
    - target stk_p1_s11_t7 (Cartesian target) at (974.53, -259.63, 694.38) mm, rotated rx -69.65 ry 82.77 rz -63.02 deg; joints [18.394, -66.335, 132.634, 26.689, -71.135, -3.627] of KR 8 1620 ARC HW
    - target stk_p1_s11_t8 (Cartesian target) at (974.75, -249.07, 694.5) mm, rotated rx -68.56 ry 83.13 rz -62.3 deg; joints [17.719, -66.514, 132.944, 25.568, -71.062, -3.549] of KR 8 1620 ARC HW
    - target stk_p1_s11_t9 (Cartesian target) at (974.97, -238.51, 694.62) mm, rotated rx -67.34 ry 83.49 rz -61.46 deg; joints [17.039, -66.687, 133.24, 24.439, -70.992, -3.473] of KR 8 1620 ARC HW
    - target stk_p1_s11_t10 (Cartesian target) at (975.19, -227.95, 694.75) mm, rotated rx -65.98 ry 83.85 rz -60.48 deg; joints [16.354, -66.853, 133.525, 23.305, -70.926, -3.397] of KR 8 1620 ARC HW
    - target stk_p1_s11_t11 (Cartesian target) at (975.41, -217.39, 694.87) mm, rotated rx -64.45 ry 84.2 rz -59.33 deg; joints [15.663, -67.012, 133.797, 22.163, -70.863, -3.323] of KR 8 1620 ARC HW
    - target stk_p1_s11_t12 (Cartesian target) at (975.63, -206.84, 695) mm, rotated rx -62.72 ry 84.55 rz -57.98 deg; joints [14.968, -67.164, 134.057, 21.016, -70.803, -3.25] of KR 8 1620 ARC HW
    - target stk_p1_s11_t13 (Cartesian target) at (975.85, -196.28, 695.12) mm, rotated rx -60.76 ry 84.89 rz -56.39 deg; joints [14.268, -67.309, 134.304, 19.863, -70.747, -3.178] of KR 8 1620 ARC HW
    - target stk_p1_s11_t14 (Cartesian target) at (976.07, -185.72, 695.24) mm, rotated rx -58.51 ry 85.23 rz -54.53 deg; joints [13.564, -67.447, 134.538, 18.704, -70.694, -3.107] of KR 8 1620 ARC HW
    - target stk_p1_s11_t15 (Cartesian target) at (976.29, -175.16, 695.37) mm, rotated rx -55.92 ry 85.56 rz -52.32 deg; joints [12.855, -67.578, 134.76, 17.54, -70.645, -3.037] of KR 8 1620 ARC HW
    - target stk_p1_s11_t16 (Cartesian target) at (976.51, -164.6, 695.49) mm, rotated rx -52.92 ry 85.88 rz -49.7 deg; joints [12.142, -67.701, 134.969, 16.371, -70.599, -2.968] of KR 8 1620 ARC HW
    - target stk_p1_s11_t17 (Cartesian target) at (976.73, -154.04, 695.61) mm, rotated rx -49.43 ry 86.18 rz -46.59 deg; joints [11.425, -67.818, 135.165, 15.197, -70.556, -2.9] of KR 8 1620 ARC HW
    - target stk_p1_s11_t18 (Cartesian target) at (976.95, -143.48, 695.74) mm, rotated rx -45.34 ry 86.48 rz -42.88 deg; joints [10.705, -67.927, 135.349, 14.018, -70.517, -2.833] of KR 8 1620 ARC HW
    - target stk_p1_s11_t19 (Cartesian target) at (977.16, -132.93, 695.86) mm, rotated rx -40.54 ry 86.74 rz -38.47 deg; joints [9.981, -68.028, 135.519, 12.836, -70.481, -2.766] of KR 8 1620 ARC HW
    - target stk_p1_s11_t20 (Cartesian target) at (977.38, -122.37, 695.98) mm, rotated rx -34.92 ry 86.99 rz -33.23 deg; joints [9.253, -68.122, 135.676, 11.649, -70.449, -2.7] of KR 8 1620 ARC HW
    - target stk_p1_s11_t21 (Cartesian target) at (977.6, -111.81, 696.11) mm, rotated rx -28.39 ry 87.2 rz -27.08 deg; joints [8.523, -68.209, 135.821, 10.458, -70.42, -2.635] of KR 8 1620 ARC HW
    - target stk_p1_s11_t22 (Cartesian target) at (977.82, -101.25, 696.23) mm, rotated rx -20.91 ry 87.36 rz -19.99 deg; joints [7.79, -68.288, 135.952, 9.265, -70.394, -2.57] of KR 8 1620 ARC HW
    - target stk_p1_s11_t23 (Cartesian target) at (978.04, -90.69, 696.35) mm, rotated rx -12.58 ry 87.48 rz -12.04 deg; joints [7.054, -68.359, 136.07, 8.068, -70.372, -2.505] of KR 8 1620 ARC HW
    - target stk_p1_s11_t24 (Cartesian target) at (978.26, -80.13, 696.48) mm, rotated rx -3.64 ry 87.54 rz -3.49 deg; joints [6.316, -68.423, 136.175, 6.868, -70.353, -2.441] of KR 8 1620 ARC HW
    - target stk_p1_s11_t25 (Cartesian target) at (978.48, -69.58, 696.6) mm, rotated rx 5.51 ry 87.54 rz 5.28 deg; joints [5.576, -68.479, 136.267, 5.666, -70.337, -2.377] of KR 8 1620 ARC HW
    - target stk_p1_s12_t0 (Cartesian target) at (980.13, -20.5, 1014.04) mm, rotated rx 167.57 ry 80.5 rz 165.34 deg; joints [2.115, -83.159, 120.084, 0.111, -27.646, -2.153] of KR 8 1620 ARC HW
    - target stk_p1_s12_t0 (Cartesian target) at (980.13, -20.5, 1014.04) mm, rotated rx 167.57 ry 80.5 rz 165.34 deg; joints [2.115, -83.159, 120.084, 0.111, -27.646, -2.153] of KR 8 1620 ARC HW
    - target stk_p1_s12_t1 (Cartesian target) at (980.35, -9.94, 1014.16) mm, rotated rx 165.31 ry 80.4 rz 162.65 deg; joints [1.372, -83.174, 120.1, -2.305, -27.661, -0.589] of KR 8 1620 ARC HW
    - target stk_p1_s12_t2 (Cartesian target) at (980.57, 0.61, 1014.29) mm, rotated rx 163.09 ry 80.29 rz 160.01 deg; joints [0.628, -83.179, 120.103, -4.717, -27.712, 0.971] of KR 8 1620 ARC HW
    - target stk_p1_s12_t3 (Cartesian target) at (980.79, 11.17, 1014.41) mm, rotated rx 160.93 ry 80.17 rz 157.42 deg; joints [-0.116, -83.174, 120.095, -7.118, -27.801, 2.52] of KR 8 1620 ARC HW
    - target stk_p1_s12_t4 (Cartesian target) at (981.01, 21.73, 1014.53) mm, rotated rx 158.82 ry 80.03 rz 154.89 deg; joints [-0.859, -83.159, 120.075, -9.502, -27.925, 4.052] of KR 8 1620 ARC HW
    - target stk_p1_s12_t5 (Cartesian target) at (981.23, 32.29, 1014.66) mm, rotated rx 156.77 ry 79.88 rz 152.42 deg; joints [-1.603, -83.133, 120.043, -11.864, -28.086, 5.563] of KR 8 1620 ARC HW
    - target stk_p1_s12_t6 (Cartesian target) at (981.45, 42.85, 1014.78) mm, rotated rx 154.79 ry 79.72 rz 150.01 deg; joints [-2.345, -83.096, 120, -14.198, -28.283, 7.046] of KR 8 1620 ARC HW
    - target stk_p1_s12_t7 (Cartesian target) at (981.66, 53.41, 1014.9) mm, rotated rx 152.87 ry 79.55 rz 147.67 deg; joints [-3.087, -83.05, 119.944, -16.5, -28.513, 8.497] of KR 8 1620 ARC HW
    - target stk_p1_s12_t8 (Cartesian target) at (981.88, 63.97, 1015.03) mm, rotated rx 151.01 ry 79.36 rz 145.39 deg; joints [-3.827, -82.993, 119.876, -18.764, -28.777, 9.911] of KR 8 1620 ARC HW
    - target stk_p1_s12_t9 (Cartesian target) at (982.1, 74.52, 1015.15) mm, rotated rx 149.23 ry 79.17 rz 143.18 deg; joints [-4.565, -82.926, 119.797, -20.987, -29.072, 11.286] of KR 8 1620 ARC HW
    - target stk_p1_s12_t10 (Cartesian target) at (982.32, 85.08, 1015.27) mm, rotated rx 147.5 ry 78.96 rz 141.04 deg; joints [-5.302, -82.848, 119.705, -23.166, -29.399, 12.617] of KR 8 1620 ARC HW
    - target stk_p1_s12_t11 (Cartesian target) at (982.54, 95.64, 1015.4) mm, rotated rx 145.85 ry 78.75 rz 138.96 deg; joints [-6.037, -82.76, 119.602, -25.297, -29.755, 13.903] of KR 8 1620 ARC HW
    - target stk_p1_s12_t12 (Cartesian target) at (982.76, 106.2, 1015.52) mm, rotated rx 144.25 ry 78.53 rz 136.94 deg; joints [-6.769, -82.663, 119.487, -27.38, -30.139, 15.14] of KR 8 1620 ARC HW
    - target stk_p1_s12_t13 (Cartesian target) at (982.98, 116.76, 1015.65) mm, rotated rx 142.72 ry 78.3 rz 134.99 deg; joints [-7.499, -82.555, 119.36, -29.411, -30.55, 16.328] of KR 8 1620 ARC HW
    - target stk_p1_s12_t14 (Cartesian target) at (983.2, 127.32, 1015.77) mm, rotated rx 141.25 ry 78.06 rz 133.1 deg; joints [-8.227, -82.437, 119.221, -31.39, -30.986, 17.465] of KR 8 1620 ARC HW
    - target stk_p1_s12_t15 (Cartesian target) at (983.42, 137.87, 1015.89) mm, rotated rx 139.84 ry 77.81 rz 131.27 deg; joints [-8.951, -82.309, 119.07, -33.315, -31.445, 18.551] of KR 8 1620 ARC HW
    - target stk_p1_s12_t16 (Cartesian target) at (983.64, 148.43, 1016.02) mm, rotated rx 138.49 ry 77.56 rz 129.5 deg; joints [-9.672, -82.171, 118.907, -35.188, -31.927, 19.586] of KR 8 1620 ARC HW
    - target stk_p1_s12_t17 (Cartesian target) at (983.86, 158.99, 1016.14) mm, rotated rx 137.19 ry 77.31 rz 127.79 deg; joints [-10.389, -82.024, 118.732, -37.007, -32.43, 20.57] of KR 8 1620 ARC HW
    - target stk_p1_s12_t18 (Cartesian target) at (984.08, 169.55, 1016.26) mm, rotated rx 135.95 ry 77.04 rz 126.13 deg; joints [-11.103, -81.867, 118.545, -38.773, -32.951, 21.503] of KR 8 1620 ARC HW
    - target stk_p1_s12_t19 (Cartesian target) at (984.3, 180.11, 1016.39) mm, rotated rx 134.76 ry 76.78 rz 124.52 deg; joints [-11.812, -81.7, 118.347, -40.487, -33.491, 22.386] of KR 8 1620 ARC HW
    - target stk_p1_s12_t20 (Cartesian target) at (984.52, 190.67, 1016.51) mm, rotated rx 133.62 ry 76.5 rz 122.96 deg; joints [-12.518, -81.523, 118.136, -42.149, -34.047, 23.22] of KR 8 1620 ARC HW
    - target stk_p1_s12_t21 (Cartesian target) at (984.73, 201.22, 1016.63) mm, rotated rx 132.52 ry 76.23 rz 121.45 deg; joints [-13.22, -81.338, 117.914, -43.761, -34.618, 24.007] of KR 8 1620 ARC HW
    - target stk_p1_s12_t22 (Cartesian target) at (984.95, 211.78, 1016.76) mm, rotated rx 131.47 ry 75.95 rz 119.98 deg; joints [-13.916, -81.143, 117.68, -45.324, -35.203, 24.748] of KR 8 1620 ARC HW
    - target stk_p1_s12_t23 (Cartesian target) at (985.17, 222.34, 1016.88) mm, rotated rx 130.46 ry 75.66 rz 118.56 deg; joints [-14.609, -80.938, 117.433, -46.84, -35.8, 25.445] of KR 8 1620 ARC HW
    - target stk_p1_s12_t24 (Cartesian target) at (985.39, 232.9, 1017) mm, rotated rx 129.49 ry 75.37 rz 117.18 deg; joints [-15.296, -80.725, 117.175, -48.308, -36.41, 26.098] of KR 8 1620 ARC HW
    - target stk_p1_s12_t25 (Cartesian target) at (985.61, 243.46, 1017.13) mm, rotated rx 128.56 ry 75.08 rz 115.84 deg; joints [-15.979, -80.503, 116.906, -49.732, -37.029, 26.71] of KR 8 1620 ARC HW
    - target stk_p1_s13_t0 (Cartesian target) at (973.55, -337.25, 1010.33) mm, rotated rx -133.48 ry 76.88 rz -123.13 deg; joints [23.081, -78.162, 114.15, 55.823, -40.139, -33.067] of KR 8 1620 ARC HW
    - target stk_p1_s13_t0 (Cartesian target) at (973.55, -337.25, 1010.33) mm, rotated rx -133.48 ry 76.88 rz -123.13 deg; joints [23.081, -78.162, 114.15, 55.823, -40.139, -33.067] of KR 8 1620 ARC HW
    - target stk_p1_s13_t1 (Cartesian target) at (973.77, -326.7, 1010.46) mm, rotated rx -134.68 ry 77.14 rz -124.73 deg; joints [22.452, -78.456, 114.516, 54.616, -39.499, -32.64] of KR 8 1620 ARC HW
    - target stk_p1_s13_t2 (Cartesian target) at (973.99, -316.14, 1010.58) mm, rotated rx -135.92 ry 77.4 rz -126.39 deg; joints [21.816, -78.743, 114.871, 53.373, -38.863, -32.182] of KR 8 1620 ARC HW
    - target stk_p1_s13_t3 (Cartesian target) at (974.21, -305.58, 1010.7) mm, rotated rx -137.22 ry 77.65 rz -128.1 deg; joints [21.175, -79.022, 115.214, 52.093, -38.233, -31.691] of KR 8 1620 ARC HW
    - target stk_p1_s13_t4 (Cartesian target) at (974.43, -295.02, 1010.83) mm, rotated rx -138.58 ry 77.9 rz -129.87 deg; joints [20.527, -79.292, 115.545, 50.773, -37.611, -31.164] of KR 8 1620 ARC HW
    - target stk_p1_s13_t5 (Cartesian target) at (974.65, -284.46, 1010.95) mm, rotated rx -139.99 ry 78.14 rz -131.69 deg; joints [19.874, -79.555, 115.865, 49.413, -36.996, -30.602] of KR 8 1620 ARC HW
    - target stk_p1_s13_t6 (Cartesian target) at (974.87, -273.9, 1011.07) mm, rotated rx -141.47 ry 78.37 rz -133.58 deg; joints [19.215, -79.809, 116.174, 48.01, -36.39, -30.001] of KR 8 1620 ARC HW
    - target stk_p1_s13_t7 (Cartesian target) at (975.09, -263.35, 1011.2) mm, rotated rx -143 ry 78.59 rz -135.53 deg; joints [18.551, -80.055, 116.471, 46.563, -35.793, -29.361] of KR 8 1620 ARC HW
    - target stk_p1_s13_t8 (Cartesian target) at (975.3, -252.79, 1011.32) mm, rotated rx -144.6 ry 78.81 rz -137.54 deg; joints [17.881, -80.293, 116.756, 45.072, -35.207, -28.678] of KR 8 1620 ARC HW
    - target stk_p1_s13_t9 (Cartesian target) at (975.52, -242.23, 1011.44) mm, rotated rx -146.26 ry 79.02 rz -139.62 deg; joints [17.206, -80.522, 117.03, 43.533, -34.633, -27.953] of KR 8 1620 ARC HW
    - target stk_p1_s13_t10 (Cartesian target) at (975.74, -231.67, 1011.57) mm, rotated rx -147.98 ry 79.22 rz -141.76 deg; joints [16.525, -80.742, 117.293, 41.946, -34.072, -27.183] of KR 8 1620 ARC HW
    - target stk_p1_s13_t11 (Cartesian target) at (975.96, -221.11, 1011.69) mm, rotated rx -149.77 ry 79.41 rz -143.97 deg; joints [15.84, -80.953, 117.543, 40.309, -33.525, -26.366] of KR 8 1620 ARC HW
    - target stk_p1_s13_t12 (Cartesian target) at (976.18, -210.55, 1011.82) mm, rotated rx -151.63 ry 79.59 rz -146.25 deg; joints [15.15, -81.156, 117.783, 38.622, -32.993, -25.502] of KR 8 1620 ARC HW
    - target stk_p1_s13_t13 (Cartesian target) at (976.4, -200, 1011.94) mm, rotated rx -153.56 ry 79.76 rz -148.59 deg; joints [14.455, -81.349, 118.01, 36.883, -32.478, -24.589] of KR 8 1620 ARC HW
    - target stk_p1_s13_t14 (Cartesian target) at (976.62, -189.44, 1012.06) mm, rotated rx -155.54 ry 79.92 rz -151 deg; joints [13.755, -81.533, 118.226, 35.092, -31.982, -23.627] of KR 8 1620 ARC HW
    - target stk_p1_s13_t15 (Cartesian target) at (976.84, -178.88, 1012.19) mm, rotated rx -157.59 ry 80.07 rz -153.47 deg; joints [13.051, -81.708, 118.43, 33.248, -31.505, -22.614] of KR 8 1620 ARC HW
    - target stk_p1_s13_t16 (Cartesian target) at (977.06, -168.32, 1012.31) mm, rotated rx -159.7 ry 80.2 rz -156 deg; joints [12.343, -81.874, 118.623, 31.351, -31.048, -21.55] of KR 8 1620 ARC HW
    - target stk_p1_s13_t17 (Cartesian target) at (977.28, -157.76, 1012.43) mm, rotated rx -161.87 ry 80.32 rz -158.59 deg; joints [11.631, -82.03, 118.803, 29.4, -30.615, -20.436] of KR 8 1620 ARC HW
    - target stk_p1_s13_t18 (Cartesian target) at (977.5, -147.2, 1012.56) mm, rotated rx -164.09 ry 80.42 rz -161.23 deg; joints [10.916, -82.176, 118.973, 27.397, -30.205, -19.271] of KR 8 1620 ARC HW
    - target stk_p1_s13_t19 (Cartesian target) at (977.72, -136.64, 1012.68) mm, rotated rx -166.36 ry 80.52 rz -163.92 deg; joints [10.196, -82.313, 119.13, 25.342, -29.82, -18.056] of KR 8 1620 ARC HW
    - target stk_p1_s13_t20 (Cartesian target) at (977.94, -126.09, 1012.8) mm, rotated rx -168.67 ry 80.59 rz -166.65 deg; joints [9.474, -82.44, 119.276, 23.237, -29.463, -16.793] of KR 8 1620 ARC HW
    - target stk_p1_s13_t21 (Cartesian target) at (978.16, -115.53, 1012.93) mm, rotated rx -171.01 ry 80.65 rz -169.42 deg; joints [8.748, -82.557, 119.41, 21.084, -29.133, -15.483] of KR 8 1620 ARC HW
    - target stk_p1_s13_t22 (Cartesian target) at (978.37, -104.97, 1013.05) mm, rotated rx -173.39 ry 80.7 rz -172.22 deg; joints [8.019, -82.665, 119.532, 18.885, -28.834, -14.129] of KR 8 1620 ARC HW
    - target stk_p1_s13_t23 (Cartesian target) at (978.59, -94.41, 1013.17) mm, rotated rx -175.78 ry 80.73 rz -175.04 deg; joints [7.288, -82.762, 119.642, 16.643, -28.566, -12.734] of KR 8 1620 ARC HW
    - target stk_p1_s13_t24 (Cartesian target) at (978.81, -83.85, 1013.3) mm, rotated rx -178.19 ry 80.75 rz -177.87 deg; joints [6.554, -82.849, 119.741, 14.361, -28.329, -11.3] of KR 8 1620 ARC HW
    - target stk_p1_s13_t25 (Cartesian target) at (979.03, -73.29, 1013.42) mm, rotated rx 179.4 ry 80.74 rz 179.29 deg; joints [5.818, -82.926, 119.828, 12.045, -28.127, -9.832] of KR 8 1620 ARC HW
    - target stk_p2_s14_t0 (Cartesian target) at (979.72, -17.78, 781.7) mm, rotated rx 108.28 ry 87.72 rz 106.1 deg; joints [1.206, -74.416, 132.822, -1.133, -57.696, -1.57] of KR 8 1620 ARC HW
    - target stk_p2_s14_t0 (Cartesian target) at (979.72, -17.78, 781.7) mm, rotated rx 108.28 ry 87.72 rz 106.1 deg; joints [1.206, -74.416, 132.822, -1.133, -57.696, -1.57] of KR 8 1620 ARC HW
    - target stk_p2_s14_t1 (Cartesian target) at (979.94, -7.22, 781.83) mm, rotated rx 105.71 ry 87.34 rz 103.14 deg; joints [0.465, -74.418, 132.813, -2.474, -57.7, -1.26] of KR 8 1620 ARC HW
    - target stk_p2_s14_t2 (Cartesian target) at (980.16, 3.34, 781.95) mm, rotated rx 103.79 ry 86.96 rz 100.82 deg; joints [-0.275, -74.412, 132.792, -3.815, -57.714, -0.95] of KR 8 1620 ARC HW
    - target stk_p2_s14_t3 (Cartesian target) at (980.38, 13.9, 782.07) mm, rotated rx 102.3 ry 86.58 rz 98.93 deg; joints [-1.015, -74.396, 132.759, -5.154, -57.738, -0.641] of KR 8 1620 ARC HW
    - target stk_p2_s14_t4 (Cartesian target) at (980.6, 24.46, 782.2) mm, rotated rx 101.1 ry 86.19 rz 97.35 deg; joints [-1.755, -74.371, 132.712, -6.492, -57.772, -0.332] of KR 8 1620 ARC HW
    - target stk_p2_s14_t5 (Cartesian target) at (980.82, 35.02, 782.32) mm, rotated rx 100.13 ry 85.81 rz 95.98 deg; joints [-2.493, -74.338, 132.654, -7.827, -57.816, -0.024] of KR 8 1620 ARC HW
    - target stk_p2_s14_t6 (Cartesian target) at (981.04, 45.58, 782.45) mm, rotated rx 99.32 ry 85.42 rz 94.78 deg; joints [-3.23, -74.296, 132.582, -9.16, -57.87, 0.283] of KR 8 1620 ARC HW
    - target stk_p2_s14_t7 (Cartesian target) at (981.26, 56.13, 782.57) mm, rotated rx 98.64 ry 85.03 rz 93.7 deg; joints [-3.966, -74.245, 132.498, -10.488, -57.935, 0.588] of KR 8 1620 ARC HW
    - target stk_p2_s14_t8 (Cartesian target) at (981.48, 66.69, 782.69) mm, rotated rx 98.06 ry 84.65 rz 92.73 deg; joints [-4.7, -74.186, 132.402, -11.813, -58.009, 0.891] of KR 8 1620 ARC HW
    - target stk_p2_s14_t9 (Cartesian target) at (981.7, 77.25, 782.82) mm, rotated rx 97.56 ry 84.26 rz 91.83 deg; joints [-5.432, -74.117, 132.293, -13.134, -58.093, 1.191] of KR 8 1620 ARC HW
    - target stk_p2_s14_t10 (Cartesian target) at (981.92, 87.81, 782.94) mm, rotated rx 97.12 ry 83.87 rz 91 deg; joints [-6.161, -74.04, 132.171, -14.449, -58.186, 1.49] of KR 8 1620 ARC HW
    - target stk_p2_s14_t11 (Cartesian target) at (982.14, 98.37, 783.06) mm, rotated rx 96.73 ry 83.48 rz 90.22 deg; joints [-6.888, -73.955, 132.037, -15.759, -58.289, 1.785] of KR 8 1620 ARC HW
    - target stk_p2_s14_t12 (Cartesian target) at (982.36, 108.93, 783.19) mm, rotated rx 96.39 ry 83.1 rz 89.48 deg; joints [-7.613, -73.861, 131.89, -17.062, -58.401, 2.078] of KR 8 1620 ARC HW
    - target stk_p2_s14_t13 (Cartesian target) at (982.58, 119.48, 783.31) mm, rotated rx 96.08 ry 82.71 rz 88.78 deg; joints [-8.334, -73.758, 131.732, -18.359, -58.522, 2.367] of KR 8 1620 ARC HW
    - target stk_p2_s14_t14 (Cartesian target) at (982.79, 130.04, 783.43) mm, rotated rx 95.8 ry 82.32 rz 88.12 deg; joints [-9.052, -73.647, 131.56, -19.649, -58.653, 2.653] of KR 8 1620 ARC HW
    - target stk_p2_s14_t15 (Cartesian target) at (983.01, 140.6, 783.56) mm, rotated rx 95.56 ry 81.94 rz 87.48 deg; joints [-9.767, -73.528, 131.377, -20.931, -58.792, 2.935] of KR 8 1620 ARC HW
    - target stk_p2_s14_t16 (Cartesian target) at (983.23, 151.16, 783.68) mm, rotated rx 95.33 ry 81.55 rz 86.86 deg; joints [-10.479, -73.4, 131.181, -22.205, -58.939, 3.213] of KR 8 1620 ARC HW
    - target stk_p2_s14_t17 (Cartesian target) at (983.45, 161.72, 783.8) mm, rotated rx 95.12 ry 81.17 rz 86.26 deg; joints [-11.186, -73.264, 130.972, -23.471, -59.095, 3.488] of KR 8 1620 ARC HW
    - target stk_p2_s14_t18 (Cartesian target) at (983.67, 172.28, 783.93) mm, rotated rx 94.94 ry 80.78 rz 85.69 deg; joints [-11.89, -73.12, 130.752, -24.728, -59.26, 3.758] of KR 8 1620 ARC HW
    - target stk_p2_s14_t19 (Cartesian target) at (983.89, 182.84, 784.05) mm, rotated rx 94.76 ry 80.4 rz 85.13 deg; joints [-12.589, -72.968, 130.519, -25.976, -59.432, 4.024] of KR 8 1620 ARC HW
    - target stk_p2_s14_t20 (Cartesian target) at (984.11, 193.39, 784.18) mm, rotated rx 94.6 ry 80.02 rz 84.58 deg; joints [-13.284, -72.809, 130.275, -27.215, -59.612, 4.286] of KR 8 1620 ARC HW
    - target stk_p2_s14_t21 (Cartesian target) at (984.33, 203.95, 784.3) mm, rotated rx 94.45 ry 79.63 rz 84.05 deg; joints [-13.974, -72.641, 130.018, -28.444, -59.8, 4.543] of KR 8 1620 ARC HW
    - target stk_p2_s14_t22 (Cartesian target) at (984.55, 214.51, 784.42) mm, rotated rx 94.32 ry 79.25 rz 83.52 deg; joints [-14.66, -72.465, 129.749, -29.663, -59.994, 4.796] of KR 8 1620 ARC HW
    - target stk_p2_s14_t23 (Cartesian target) at (984.77, 225.07, 784.55) mm, rotated rx 94.19 ry 78.87 rz 83.01 deg; joints [-15.34, -72.282, 129.468, -30.871, -60.196, 5.045] of KR 8 1620 ARC HW
    - target stk_p2_s14_t24 (Cartesian target) at (984.99, 235.63, 784.67) mm, rotated rx 94.07 ry 78.49 rz 82.51 deg; joints [-16.016, -72.091, 129.175, -32.069, -60.405, 5.289] of KR 8 1620 ARC HW
    - target stk_p2_s14_t25 (Cartesian target) at (985.21, 246.19, 784.79) mm, rotated rx 93.96 ry 78.11 rz 82.01 deg; joints [-16.687, -71.893, 128.871, -33.256, -60.621, 5.529] of KR 8 1620 ARC HW
    - target stk_p2_s15_t0 (Cartesian target) at (973.14, -334.53, 778) mm, rotated rx -93.43 ry 80.49 rz -83.89 deg; joints [22.329, -70.438, 127.302, 36.756, -61.79, -9.596] of KR 8 1620 ARC HW
    - target stk_p2_s15_t0 (Cartesian target) at (973.14, -334.53, 778) mm, rotated rx -93.43 ry 80.49 rz -83.89 deg; joints [22.329, -70.438, 127.302, 36.756, -61.79, -9.596] of KR 8 1620 ARC HW
    - target stk_p2_s15_t1 (Cartesian target) at (973.36, -323.97, 778.12) mm, rotated rx -93.6 ry 80.86 rz -84.44 deg; joints [21.689, -70.682, 127.661, 35.624, -61.549, -9.389] of KR 8 1620 ARC HW
    - target stk_p2_s15_t2 (Cartesian target) at (973.58, -313.41, 778.25) mm, rotated rx -93.79 ry 81.24 rz -85.01 deg; joints [21.042, -70.919, 128.008, 34.48, -61.313, -9.178] of KR 8 1620 ARC HW
    - target stk_p2_s15_t3 (Cartesian target) at (973.8, -302.85, 778.37) mm, rotated rx -94 ry 81.62 rz -85.6 deg; joints [20.39, -71.15, 128.344, 33.326, -61.083, -8.963] of KR 8 1620 ARC HW
    - target stk_p2_s15_t4 (Cartesian target) at (974.02, -292.29, 778.49) mm, rotated rx -94.23 ry 82.01 rz -86.21 deg; joints [19.732, -71.373, 128.667, 32.16, -60.858, -8.742] of KR 8 1620 ARC HW
    - target stk_p2_s15_t5 (Cartesian target) at (974.24, -281.74, 778.62) mm, rotated rx -94.48 ry 82.39 rz -86.85 deg; joints [19.069, -71.589, 128.979, 30.983, -60.639, -8.518] of KR 8 1620 ARC HW
    - target stk_p2_s15_t6 (Cartesian target) at (974.46, -271.18, 778.74) mm, rotated rx -94.76 ry 82.77 rz -87.51 deg; joints [18.401, -71.798, 129.28, 29.795, -60.426, -8.288] of KR 8 1620 ARC HW
    - target stk_p2_s15_t7 (Cartesian target) at (974.68, -260.62, 778.86) mm, rotated rx -95.06 ry 83.15 rz -88.21 deg; joints [17.727, -72, 129.568, 28.596, -60.22, -8.054] of KR 8 1620 ARC HW
    - target stk_p2_s15_t8 (Cartesian target) at (974.9, -250.06, 778.99) mm, rotated rx -95.41 ry 83.54 rz -88.94 deg; joints [17.048, -72.194, 129.844, 27.388, -60.02, -7.815] of KR 8 1620 ARC HW
    - target stk_p2_s15_t9 (Cartesian target) at (975.12, -239.5, 779.11) mm, rotated rx -95.8 ry 83.92 rz -89.72 deg; joints [16.365, -72.381, 130.109, 26.169, -59.826, -7.572] of KR 8 1620 ARC HW
    - target stk_p2_s15_t10 (Cartesian target) at (975.34, -228.94, 779.23) mm, rotated rx -96.24 ry 84.3 rz -90.55 deg; joints [15.676, -72.56, 130.361, 24.94, -59.64, -7.324] of KR 8 1620 ARC HW
    - target stk_p2_s15_t11 (Cartesian target) at (975.56, -218.39, 779.36) mm, rotated rx -96.75 ry 84.69 rz -91.45 deg; joints [14.983, -72.731, 130.601, 23.701, -59.461, -7.071] of KR 8 1620 ARC HW
    - target stk_p2_s15_t12 (Cartesian target) at (975.78, -207.83, 779.48) mm, rotated rx -97.34 ry 85.07 rz -92.43 deg; joints [14.285, -72.895, 130.83, 22.453, -59.289, -6.814] of KR 8 1620 ARC HW
    - target stk_p2_s15_t13 (Cartesian target) at (976, -197.27, 779.6) mm, rotated rx -98.03 ry 85.46 rz -93.5 deg; joints [13.584, -73.05, 131.046, 21.197, -59.125, -6.552] of KR 8 1620 ARC HW
    - target stk_p2_s15_t14 (Cartesian target) at (976.22, -186.71, 779.73) mm, rotated rx -98.84 ry 85.84 rz -94.71 deg; joints [12.878, -73.198, 131.249, 19.931, -58.969, -6.285] of KR 8 1620 ARC HW
    - target stk_p2_s15_t15 (Cartesian target) at (976.43, -176.15, 779.85) mm, rotated rx -99.82 ry 86.23 rz -96.09 deg; joints [12.168, -73.338, 131.441, 18.658, -58.821, -6.015] of KR 8 1620 ARC HW
    - target stk_p2_s15_t16 (Cartesian target) at (976.65, -165.59, 779.97) mm, rotated rx -101.03 ry 86.61 rz -97.68 deg; joints [11.454, -73.469, 131.62, 17.376, -58.682, -5.74] of KR 8 1620 ARC HW
    - target stk_p2_s15_t17 (Cartesian target) at (976.87, -155.03, 780.1) mm, rotated rx -102.55 ry 86.99 rz -99.59 deg; joints [10.738, -73.592, 131.787, 16.087, -58.55, -5.461] of KR 8 1620 ARC HW
    - target stk_p2_s15_t18 (Cartesian target) at (977.09, -144.48, 780.22) mm, rotated rx -104.5 ry 87.37 rz -101.94 deg; joints [10.017, -73.707, 131.942, 14.791, -58.428, -5.178] of KR 8 1620 ARC HW
    - target stk_p2_s15_t19 (Cartesian target) at (977.31, -133.92, 780.35) mm, rotated rx -107.11 ry 87.75 rz -104.94 deg; joints [9.294, -73.814, 132.084, 13.488, -58.315, -4.892] of KR 8 1620 ARC HW
    - target stk_p2_s15_t20 (Cartesian target) at (977.53, -123.36, 780.47) mm, rotated rx -110.75 ry 88.12 rz -108.98 deg; joints [8.568, -73.912, 132.214, 12.179, -58.21, -4.602] of KR 8 1620 ARC HW
    - target stk_p2_s15_t21 (Cartesian target) at (977.75, -112.8, 780.59) mm, rotated rx -116.14 ry 88.47 rz -114.76 deg; joints [7.839, -74.001, 132.331, 10.864, -58.115, -4.309] of KR 8 1620 ARC HW
    - target stk_p2_s15_t22 (Cartesian target) at (977.97, -102.24, 780.72) mm, rotated rx -124.7 ry 88.81 rz -123.72 deg; joints [7.108, -74.082, 132.436, 9.545, -58.029, -4.013] of KR 8 1620 ARC HW
    - target stk_p2_s15_t23 (Cartesian target) at (978.19, -91.68, 780.84) mm, rotated rx -139.34 ry 89.1 rz -138.75 deg; joints [6.375, -74.155, 132.528, 8.22, -57.953, -3.714] of KR 8 1620 ARC HW
    - target stk_p2_s15_t24 (Cartesian target) at (978.41, -81.13, 780.96) mm, rotated rx -164.29 ry 89.29 rz -164.09 deg; joints [5.64, -74.218, 132.608, 6.892, -57.886, -3.413] of KR 8 1620 ARC HW
    - target stk_p2_s15_t25 (Cartesian target) at (978.63, -70.57, 781.09) mm, rotated rx 163.91 ry 89.28 rz 163.71 deg; joints [4.904, -74.273, 132.675, 5.56, -57.83, -3.11] of KR 8 1620 ARC HW
    - target stk_p2_s16_t0 (Cartesian target) at (979.91, -19.01, 887.31) mm, rotated rx 155.49 ry 84.91 rz 153.28 deg; joints [1.294, -79.362, 127.375, -1.196, -43.385, -1.316] of KR 8 1620 ARC HW
    - target stk_p2_s16_t0 (Cartesian target) at (979.91, -19.01, 887.31) mm, rotated rx 155.49 ry 84.91 rz 153.28 deg; joints [1.294, -79.362, 127.375, -1.196, -43.385, -1.316] of KR 8 1620 ARC HW
    - target stk_p2_s16_t1 (Cartesian target) at (980.13, -8.46, 887.43) mm, rotated rx 151.63 ry 84.73 rz 149.02 deg; joints [0.555, -79.364, 127.367, -2.838, -43.398, -0.606] of KR 8 1620 ARC HW
    - target stk_p2_s16_t2 (Cartesian target) at (980.35, 2.1, 887.56) mm, rotated rx 148.04 ry 84.53 rz 145.02 deg; joints [-0.183, -79.356, 127.347, -4.478, -43.431, 0.101] of KR 8 1620 ARC HW
    - target stk_p2_s16_t3 (Cartesian target) at (980.57, 12.66, 887.68) mm, rotated rx 144.71 ry 84.31 rz 141.28 deg; joints [-0.922, -79.338, 127.316, -6.115, -43.483, 0.807] of KR 8 1620 ARC HW
    - target stk_p2_s16_t4 (Cartesian target) at (980.79, 23.22, 887.81) mm, rotated rx 141.65 ry 84.07 rz 137.81 deg; joints [-1.659, -79.311, 127.272, -7.748, -43.554, 1.508] of KR 8 1620 ARC HW
    - target stk_p2_s16_t5 (Cartesian target) at (981, 33.78, 887.93) mm, rotated rx 138.83 ry 83.82 rz 134.58 deg; joints [-2.396, -79.274, 127.216, -9.374, -43.645, 2.204] of KR 8 1620 ARC HW
    - target stk_p2_s16_t6 (Cartesian target) at (981.22, 44.34, 888.05) mm, rotated rx 136.23 ry 83.55 rz 131.58 deg; joints [-3.131, -79.228, 127.148, -10.993, -43.754, 2.894] of KR 8 1620 ARC HW
    - target stk_p2_s16_t7 (Cartesian target) at (981.44, 54.89, 888.18) mm, rotated rx 133.85 ry 83.27 rz 128.79 deg; joints [-3.865, -79.172, 127.068, -12.604, -43.882, 3.577] of KR 8 1620 ARC HW
    - target stk_p2_s16_t8 (Cartesian target) at (981.66, 65.45, 888.3) mm, rotated rx 131.66 ry 82.98 rz 126.19 deg; joints [-4.597, -79.107, 126.976, -14.204, -44.029, 4.251] of KR 8 1620 ARC HW
    - target stk_p2_s16_t9 (Cartesian target) at (981.88, 76.01, 888.42) mm, rotated rx 129.65 ry 82.68 rz 123.78 deg; joints [-5.327, -79.032, 126.871, -15.793, -44.193, 4.915] of KR 8 1620 ARC HW
    - target stk_p2_s16_t10 (Cartesian target) at (982.1, 86.57, 888.55) mm, rotated rx 127.8 ry 82.38 rz 121.52 deg; joints [-6.055, -78.947, 126.755, -17.37, -44.375, 5.569] of KR 8 1620 ARC HW
    - target stk_p2_s16_t11 (Cartesian target) at (982.32, 97.13, 888.67) mm, rotated rx 126.1 ry 82.06 rz 119.41 deg; joints [-6.781, -78.854, 126.627, -18.933, -44.574, 6.211] of KR 8 1620 ARC HW
    - target stk_p2_s16_t12 (Cartesian target) at (982.54, 107.69, 888.79) mm, rotated rx 124.52 ry 81.75 rz 117.43 deg; joints [-7.504, -78.75, 126.487, -20.482, -44.79, 6.841] of KR 8 1620 ARC HW
    - target stk_p2_s16_t13 (Cartesian target) at (982.76, 118.24, 888.92) mm, rotated rx 123.07 ry 81.42 rz 115.57 deg; joints [-8.224, -78.638, 126.335, -22.015, -45.022, 7.458] of KR 8 1620 ARC HW
    - target stk_p2_s16_t14 (Cartesian target) at (982.98, 128.8, 889.04) mm, rotated rx 121.72 ry 81.09 rz 113.82 deg; joints [-8.941, -78.517, 126.171, -23.531, -45.27, 8.061] of KR 8 1620 ARC HW
    - target stk_p2_s16_t15 (Cartesian target) at (983.2, 139.36, 889.16) mm, rotated rx 120.47 ry 80.76 rz 112.16 deg; joints [-9.655, -78.386, 125.995, -25.031, -45.533, 8.65] of KR 8 1620 ARC HW
    - target stk_p2_s16_t16 (Cartesian target) at (983.42, 149.92, 889.29) mm, rotated rx 119.31 ry 80.42 rz 110.6 deg; joints [-10.365, -78.247, 125.807, -26.513, -45.811, 9.224] of KR 8 1620 ARC HW
    - target stk_p2_s16_t17 (Cartesian target) at (983.64, 160.48, 889.41) mm, rotated rx 118.23 ry 80.09 rz 109.12 deg; joints [-11.071, -78.098, 125.608, -27.977, -46.102, 9.783] of KR 8 1620 ARC HW
    - target stk_p2_s16_t18 (Cartesian target) at (983.86, 171.04, 889.53) mm, rotated rx 117.22 ry 79.74 rz 107.71 deg; joints [-11.774, -77.941, 125.396, -29.421, -46.408, 10.326] of KR 8 1620 ARC HW
    - target stk_p2_s16_t19 (Cartesian target) at (984.08, 181.6, 889.66) mm, rotated rx 116.28 ry 79.4 rz 106.36 deg; joints [-12.472, -77.775, 125.173, -30.846, -46.726, 10.854] of KR 8 1620 ARC HW
    - target stk_p2_s16_t20 (Cartesian target) at (984.29, 192.15, 889.78) mm, rotated rx 115.4 ry 79.05 rz 105.08 deg; joints [-13.166, -77.6, 124.938, -32.252, -47.057, 11.365] of KR 8 1620 ARC HW
    - target stk_p2_s16_t21 (Cartesian target) at (984.51, 202.71, 889.91) mm, rotated rx 114.57 ry 78.71 rz 103.86 deg; joints [-13.855, -77.417, 124.691, -33.637, -47.4, 11.86] of KR 8 1620 ARC HW
    - target stk_p2_s16_t22 (Cartesian target) at (984.73, 213.27, 890.03) mm, rotated rx 113.8 ry 78.36 rz 102.68 deg; joints [-14.54, -77.225, 124.433, -35.002, -47.754, 12.34] of KR 8 1620 ARC HW
    - target stk_p2_s16_t23 (Cartesian target) at (984.95, 223.83, 890.15) mm, rotated rx 113.07 ry 78.01 rz 101.56 deg; joints [-15.22, -77.026, 124.162, -36.347, -48.118, 12.803] of KR 8 1620 ARC HW
    - target stk_p2_s16_t24 (Cartesian target) at (985.17, 234.39, 890.28) mm, rotated rx 112.38 ry 77.66 rz 100.47 deg; joints [-15.895, -76.817, 123.88, -37.671, -48.493, 13.249] of KR 8 1620 ARC HW
    - target stk_p2_s16_t25 (Cartesian target) at (985.39, 244.95, 890.4) mm, rotated rx 111.73 ry 77.31 rz 99.43 deg; joints [-16.565, -76.601, 123.587, -38.974, -48.877, 13.68] of KR 8 1620 ARC HW
    - target stk_p2_s17_t0 (Cartesian target) at (973.33, -335.77, 883.6) mm, rotated rx -114.99 ry 79.49 rz -105.08 deg; joints [22.354, -75.043, 122.053, 42.916, -50.688, -18.211] of KR 8 1620 ARC HW
    - target stk_p2_s17_t0 (Cartesian target) at (973.33, -335.77, 883.6) mm, rotated rx -114.99 ry 79.49 rz -105.08 deg; joints [22.354, -75.043, 122.053, 42.916, -50.688, -18.211] of KR 8 1620 ARC HW
    - target stk_p2_s17_t1 (Cartesian target) at (973.55, -325.21, 883.73) mm, rotated rx -115.94 ry 79.83 rz -106.42 deg; joints [21.715, -75.309, 122.4, 41.707, -50.272, -17.858] of KR 8 1620 ARC HW
    - target stk_p2_s17_t2 (Cartesian target) at (973.77, -314.65, 883.85) mm, rotated rx -116.95 ry 80.17 rz -107.82 deg; joints [21.071, -75.566, 122.736, 40.478, -49.864, -17.49] of KR 8 1620 ARC HW
    - target stk_p2_s17_t3 (Cartesian target) at (973.99, -304.09, 883.98) mm, rotated rx -118.03 ry 80.5 rz -109.3 deg; joints [20.42, -75.817, 123.061, 39.229, -49.463, -17.106] of KR 8 1620 ARC HW
    - target stk_p2_s17_t4 (Cartesian target) at (974.21, -293.53, 884.1) mm, rotated rx -119.2 ry 80.83 rz -110.87 deg; joints [19.765, -76.059, 123.374, 37.96, -49.07, -16.708] of KR 8 1620 ARC HW
    - target stk_p2_s17_t5 (Cartesian target) at (974.43, -282.98, 884.22) mm, rotated rx -120.45 ry 81.16 rz -112.52 deg; joints [19.104, -76.294, 123.675, 36.67, -48.686, -16.294] of KR 8 1620 ARC HW
    - target stk_p2_s17_t6 (Cartesian target) at (974.64, -272.42, 884.35) mm, rotated rx -121.8 ry 81.48 rz -114.27 deg; joints [18.437, -76.521, 123.965, 35.36, -48.31, -15.864] of KR 8 1620 ARC HW
    - target stk_p2_s17_t7 (Cartesian target) at (974.86, -261.86, 884.47) mm, rotated rx -123.27 ry 81.8 rz -116.13 deg; joints [17.765, -76.74, 124.243, 34.03, -47.944, -15.419] of KR 8 1620 ARC HW
    - target stk_p2_s17_t8 (Cartesian target) at (975.08, -251.3, 884.59) mm, rotated rx -124.85 ry 82.12 rz -118.11 deg; joints [17.089, -76.951, 124.509, 32.679, -47.588, -14.957] of KR 8 1620 ARC HW
    - target stk_p2_s17_t9 (Cartesian target) at (975.3, -240.74, 884.72) mm, rotated rx -126.56 ry 82.43 rz -120.23 deg; joints [16.407, -77.154, 124.764, 31.308, -47.242, -14.479] of KR 8 1620 ARC HW
    - target stk_p2_s17_t10 (Cartesian target) at (975.52, -230.18, 884.84) mm, rotated rx -128.42 ry 82.73 rz -122.49 deg; joints [15.721, -77.349, 125.007, 29.917, -46.908, -13.984] of KR 8 1620 ARC HW
    - target stk_p2_s17_t11 (Cartesian target) at (975.74, -219.62, 884.96) mm, rotated rx -130.44 ry 83.02 rz -124.91 deg; joints [15.03, -77.535, 125.239, 28.506, -46.585, -13.474] of KR 8 1620 ARC HW
    - target stk_p2_s17_t12 (Cartesian target) at (975.96, -209.07, 885.09) mm, rotated rx -132.64 ry 83.31 rz -127.51 deg; joints [14.334, -77.713, 125.459, 27.075, -46.275, -12.948] of KR 8 1620 ARC HW
    - target stk_p2_s17_t13 (Cartesian target) at (976.18, -198.51, 885.21) mm, rotated rx -135.03 ry 83.58 rz -130.31 deg; joints [13.635, -77.882, 125.666, 25.626, -45.978, -12.405] of KR 8 1620 ARC HW
    - target stk_p2_s17_t14 (Cartesian target) at (976.4, -187.95, 885.33) mm, rotated rx -137.64 ry 83.85 rz -133.32 deg; joints [12.931, -78.043, 125.862, 24.158, -45.694, -11.848] of KR 8 1620 ARC HW
    - target stk_p2_s17_t15 (Cartesian target) at (976.62, -177.39, 885.46) mm, rotated rx -140.47 ry 84.1 rz -136.56 deg; joints [12.223, -78.194, 126.047, 22.671, -45.424, -11.274] of KR 8 1620 ARC HW
    - target stk_p2_s17_t16 (Cartesian target) at (976.84, -166.83, 885.58) mm, rotated rx -143.55 ry 84.33 rz -140.04 deg; joints [11.512, -78.337, 126.219, 21.168, -45.168, -10.686] of KR 8 1620 ARC HW
    - target stk_p2_s17_t17 (Cartesian target) at (977.06, -156.27, 885.71) mm, rotated rx -146.89 ry 84.55 rz -143.79 deg; joints [10.797, -78.471, 126.379, 19.647, -44.928, -10.084] of KR 8 1620 ARC HW
    - target stk_p2_s17_t18 (Cartesian target) at (977.28, -145.72, 885.83) mm, rotated rx -150.5 ry 84.75 rz -147.8 deg; joints [10.079, -78.596, 126.528, 18.11, -44.704, -9.468] of KR 8 1620 ARC HW
    - target stk_p2_s17_t19 (Cartesian target) at (977.5, -135.16, 885.95) mm, rotated rx -154.37 ry 84.92 rz -152.08 deg; joints [9.358, -78.711, 126.665, 16.559, -44.495, -8.839] of KR 8 1620 ARC HW
    - target stk_p2_s17_t20 (Cartesian target) at (977.72, -124.6, 886.08) mm, rotated rx -158.5 ry 85.07 rz -156.62 deg; joints [8.635, -78.818, 126.789, 14.992, -44.304, -8.197] of KR 8 1620 ARC HW
    - target stk_p2_s17_t21 (Cartesian target) at (977.93, -114.04, 886.2) mm, rotated rx -162.88 ry 85.2 rz -161.4 deg; joints [7.908, -78.915, 126.902, 13.413, -44.129, -7.544] of KR 8 1620 ARC HW
    - target stk_p2_s17_t22 (Cartesian target) at (978.15, -103.48, 886.32) mm, rotated rx -167.46 ry 85.29 rz -166.39 deg; joints [7.179, -79.002, 127.003, 11.822, -43.972, -6.88] of KR 8 1620 ARC HW
    - target stk_p2_s17_t23 (Cartesian target) at (978.37, -92.92, 886.45) mm, rotated rx -172.19 ry 85.36 rz -171.54 deg; joints [6.449, -79.081, 127.091, 10.219, -43.833, -6.207] of KR 8 1620 ARC HW
    - target stk_p2_s17_t24 (Cartesian target) at (978.59, -82.37, 886.57) mm, rotated rx -177.03 ry 85.39 rz -176.78 deg; joints [5.716, -79.15, 127.168, 8.607, -43.712, -5.524] of KR 8 1620 ARC HW
    - target stk_p2_s17_t25 (Cartesian target) at (978.81, -71.81, 886.69) mm, rotated rx 178.1 ry 85.39 rz 177.94 deg; joints [4.981, -79.209, 127.233, 6.986, -43.61, -4.835] of KR 8 1620 ARC HW
    - target stk_p2_s18_t0 (Cartesian target) at (972.96, -333.29, 672.39) mm, rotated rx -70.7 ry 80 rz -61.52 deg; joints [22.288, -64.515, 131.191, 33.207, -73.534, -3.092] of KR 8 1620 ARC HW
    - target stk_p2_s18_t0 (Cartesian target) at (972.96, -333.29, 672.39) mm, rotated rx -70.7 ry 80 rz -61.52 deg; joints [22.288, -64.515, 131.191, 33.207, -73.534, -3.092] of KR 8 1620 ARC HW
    - target stk_p2_s18_t1 (Cartesian target) at (973.18, -322.73, 672.51) mm, rotated rx -69.97 ry 80.35 rz -61.16 deg; joints [21.646, -64.728, 131.56, 32.142, -73.447, -3.03] of KR 8 1620 ARC HW
    - target stk_p2_s18_t2 (Cartesian target) at (973.4, -312.17, 672.64) mm, rotated rx -69.18 ry 80.71 rz -60.73 deg; joints [20.998, -64.936, 131.918, 31.07, -73.363, -2.97] of KR 8 1620 ARC HW
    - target stk_p2_s18_t3 (Cartesian target) at (973.62, -301.61, 672.76) mm, rotated rx -68.32 ry 81.07 rz -60.25 deg; joints [20.344, -65.137, 132.264, 29.99, -73.282, -2.912] of KR 8 1620 ARC HW
    - target stk_p2_s18_t4 (Cartesian target) at (973.84, -291.05, 672.89) mm, rotated rx -67.39 ry 81.42 rz -59.69 deg; joints [19.685, -65.331, 132.598, 28.904, -73.204, -2.856] of KR 8 1620 ARC HW
    - target stk_p2_s18_t5 (Cartesian target) at (974.06, -280.5, 673.01) mm, rotated rx -66.37 ry 81.78 rz -59.05 deg; joints [19.02, -65.52, 132.92, 27.81, -73.128, -2.802] of KR 8 1620 ARC HW
    - target stk_p2_s18_t6 (Cartesian target) at (974.28, -269.94, 673.13) mm, rotated rx -65.27 ry 82.13 rz -58.31 deg; joints [18.35, -65.702, 133.23, 26.71, -73.056, -2.75] of KR 8 1620 ARC HW
